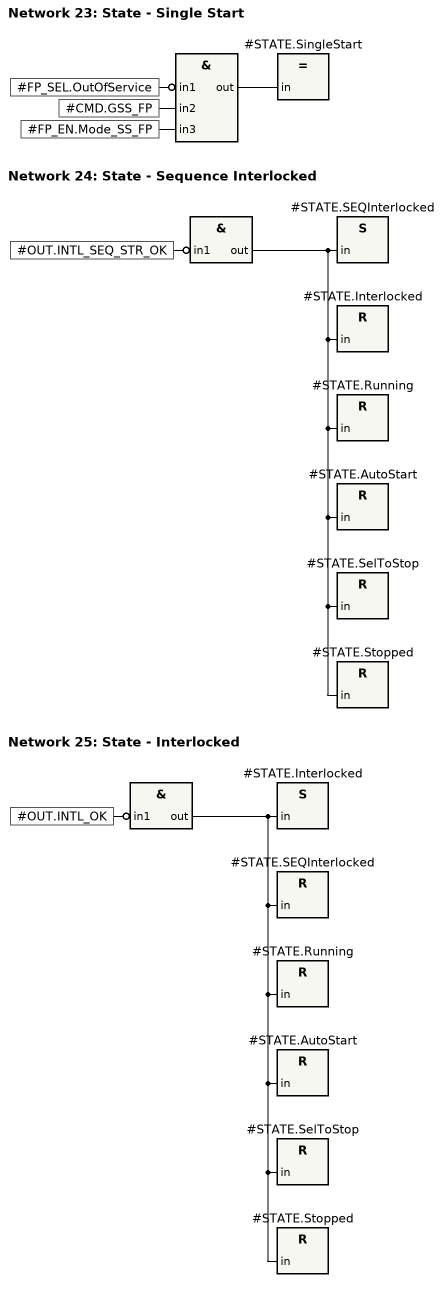
   #STATE.SingleStart := NOT #FP_SEL.OutOfService AND #CMD.GSS_FP AND #FP_EN.Mode_SS_FP;
END_REGION

REGION Network 24: State - Sequence Interlocked
   // Build 3 - SA added
   IF NOT #OUT.INTL_SEQ_STR_OK THEN
       #STATE.SEQInterlocked := TRUE;
       #STATE.Interlocked := FALSE;
       #STATE.Running := FALSE;
       #STATE.AutoStart := FALSE;
       #STATE.SelToStop := FALSE;
       #STATE.Stopped := FALSE;
   END_IF;
END_REGION

REGION Network 25: State - Interlocked
   IF NOT #OUT.INTL_OK THEN
       #STATE.Interlocked := TRUE;
       #STATE.SEQInterlocked := FALSE;
       #STATE.Running := FALSE;
       #STATE.AutoStart := FALSE;
       #STATE.SelToStop := FALSE;
       #STATE.Stopped := FALSE;
   END_IF;
END_REGION

REGION Network 26: Set Output Command for Programs
   // Start command
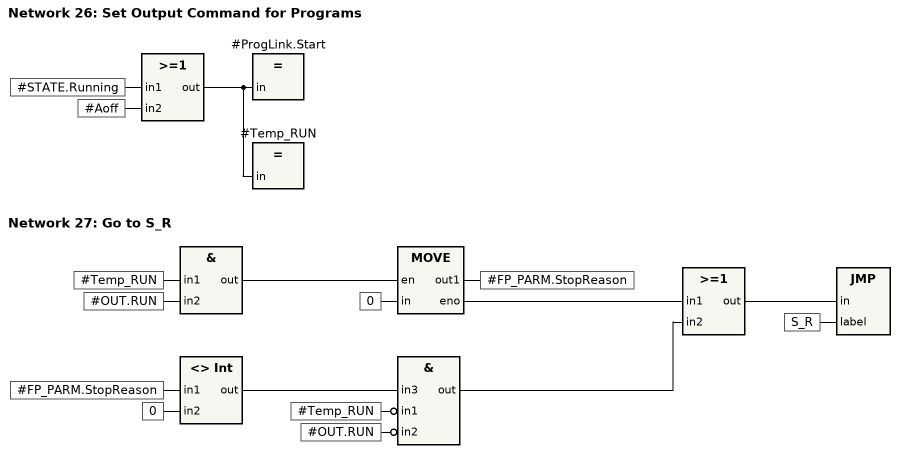
   #ProgLink.Start := #STATE.Running OR #Aoff;
   #Temp_RUN := #ProgLink.Start;
END_REGION

REGION Network 27: Go to S_R
   // ENO of a box is taken as its EN; it also drops when the box reports an error
   #_w1 := #Temp_RUN AND #OUT.RUN;
   IF #_w1 THEN #FP_PARM.StopReason := 0; END_IF;
   IF #_w1 OR ((#FP_PARM.StopReason <> 0) AND NOT #Temp_RUN AND NOT #OUT.RUN) THEN GOTO S_R; END_IF;
END_REGION

REGION Network 28: Stop Reason
   // 0=In Operation
   // 1=Normal Stop
   // 2=Quick Stop
   // 3=Faceplate Stop
   // 6=Quick Stop From Unit Faceplate
   // 9=Sequence Interlock
   // 10=Interlock
   // 12=Emergency Stop
   // 13=Auto Start
   // 99=Unknown Reason
   // 
   // 
   // Build 003-11 Aug 2021- SURAM-IN- Interval Start Stop Reason Added
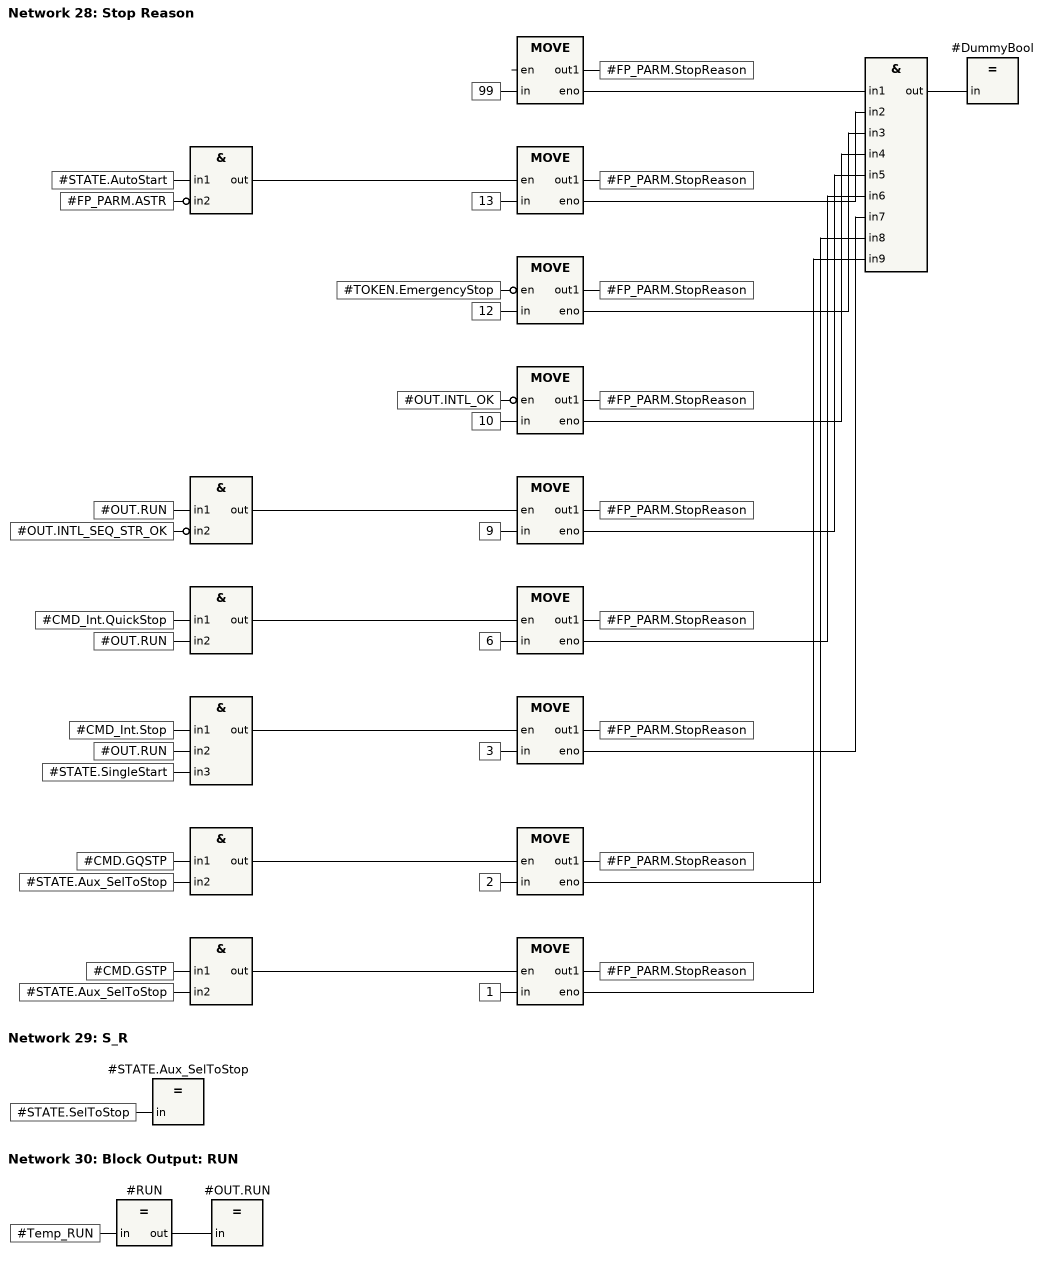
   // ENO of a box is taken as its EN; it also drops when the box reports an error
   #FP_PARM.StopReason := 99;
   #_w1 := #STATE.AutoStart AND NOT #FP_PARM.ASTR;
   IF #_w1 THEN #FP_PARM.StopReason := 13; END_IF;
   IF NOT #TOKEN.EmergencyStop THEN #FP_PARM.StopReason := 12; END_IF;
   IF NOT #OUT.INTL_OK THEN #FP_PARM.StopReason := 10; END_IF;
   #_w2 := #OUT.RUN AND NOT #OUT.INTL_SEQ_STR_OK;
   IF #_w2 THEN #FP_PARM.StopReason := 9; END_IF;
   #_w3 := #CMD_Int.QuickStop AND #OUT.RUN;
   IF #_w3 THEN #FP_PARM.StopReason := 6; END_IF;
   #_w4 := #CMD_Int.Stop AND #OUT.RUN AND #STATE.SingleStart;
   IF #_w4 THEN #FP_PARM.StopReason := 3; END_IF;
   #_w5 := #CMD.GQSTP AND #STATE.Aux_SelToStop;
   IF #_w5 THEN #FP_PARM.StopReason := 2; END_IF;
   #_w6 := #CMD.GSTP AND #STATE.Aux_SelToStop;
   IF #_w6 THEN #FP_PARM.StopReason := 1; END_IF;
   #DummyBool := #_w1 AND NOT #TOKEN.EmergencyStop AND NOT #OUT.INTL_OK AND #_w2 AND #_w3 AND #_w4 AND #_w5 AND #_w6;
END_REGION

REGION Network 29: S_R
   S_R:
   #STATE.Aux_SelToStop := #STATE.SelToStop;
END_REGION

REGION Network 30: Block Output: RUN
   #RUN := #Temp_RUN;
   #OUT.RUN := #Temp_RUN;
END_REGION

REGION Network 31: Reset Commands
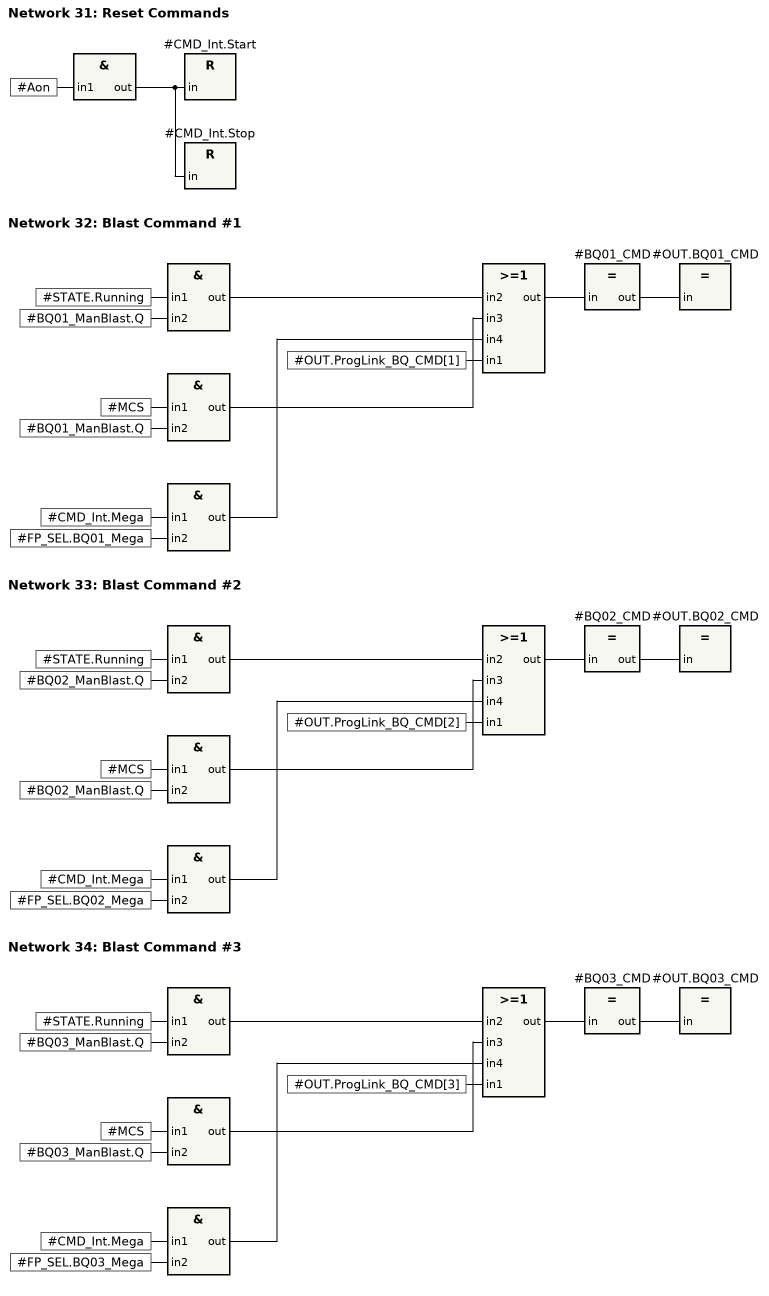
   IF #Aon THEN
       #CMD_Int.Start := FALSE;
       #CMD_Int.Stop := FALSE;
   END_IF;
END_REGION

REGION Network 32: Blast Command #1
   #BQ01_CMD := (#STATE.Running AND #BQ01_ManBlast.Q) OR (#MCS AND #BQ01_ManBlast.Q) OR (#CMD_Int.Mega AND #FP_SEL.BQ01_Mega) OR #OUT.ProgLink_BQ_CMD[1];
   #OUT.BQ01_CMD := #BQ01_CMD;
END_REGION

REGION Network 33: Blast Command #2
   #BQ02_CMD := (#STATE.Running AND #BQ02_ManBlast.Q) OR (#MCS AND #BQ02_ManBlast.Q) OR (#CMD_Int.Mega AND #FP_SEL.BQ02_Mega) OR #OUT.ProgLink_BQ_CMD[2];
   #OUT.BQ02_CMD := #BQ02_CMD;
END_REGION

REGION Network 34: Blast Command #3
   #BQ03_CMD := (#STATE.Running AND #BQ03_ManBlast.Q) OR (#MCS AND #BQ03_ManBlast.Q) OR (#CMD_Int.Mega AND #FP_SEL.BQ03_Mega) OR #OUT.ProgLink_BQ_CMD[3];
   #OUT.BQ03_CMD := #BQ03_CMD;
END_REGION

REGION Network 35: Blast Command #4
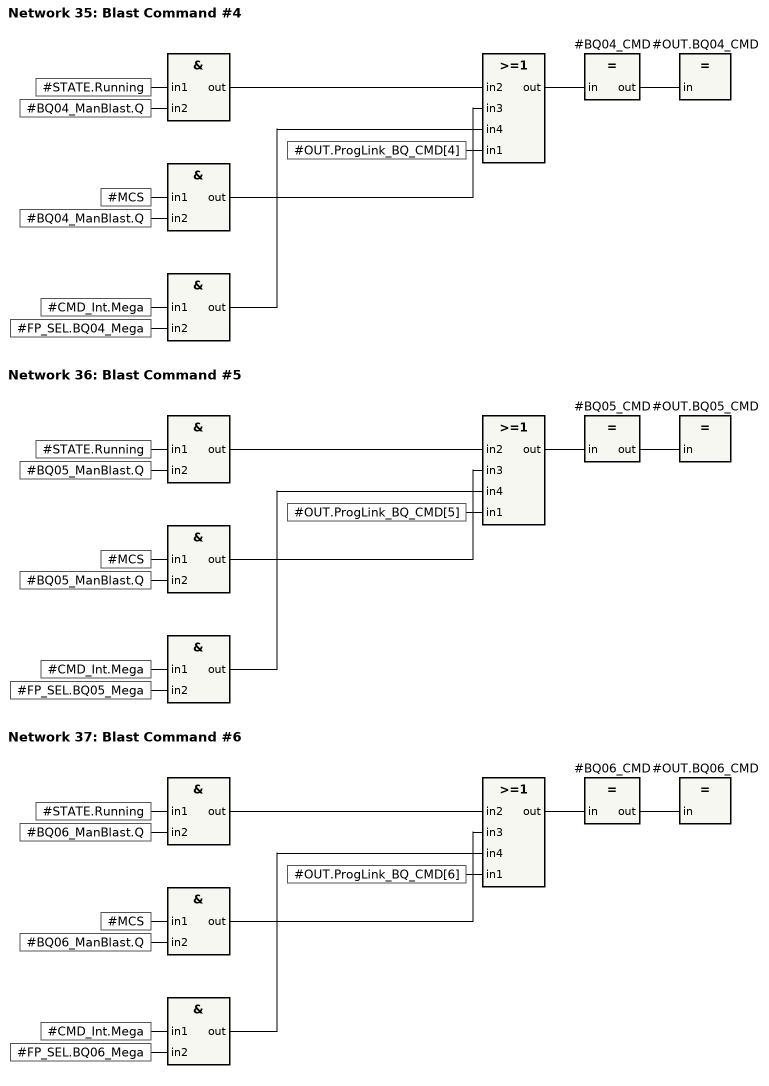
   #BQ04_CMD := (#STATE.Running AND #BQ04_ManBlast.Q) OR (#MCS AND #BQ04_ManBlast.Q) OR (#CMD_Int.Mega AND #FP_SEL.BQ04_Mega) OR #OUT.ProgLink_BQ_CMD[4];
   #OUT.BQ04_CMD := #BQ04_CMD;
END_REGION

REGION Network 36: Blast Command #5
   #BQ05_CMD := (#STATE.Running AND #BQ05_ManBlast.Q) OR (#MCS AND #BQ05_ManBlast.Q) OR (#CMD_Int.Mega AND #FP_SEL.BQ05_Mega) OR #OUT.ProgLink_BQ_CMD[5];
   #OUT.BQ05_CMD := #BQ05_CMD;
END_REGION

REGION Network 37: Blast Command #6
   #BQ06_CMD := (#STATE.Running AND #BQ06_ManBlast.Q) OR (#MCS AND #BQ06_ManBlast.Q) OR (#CMD_Int.Mega AND #FP_SEL.BQ06_Mega) OR #OUT.ProgLink_BQ_CMD[6];
   #OUT.BQ06_CMD := #BQ06_CMD;
END_REGION

REGION Network 38: Blast Command #7
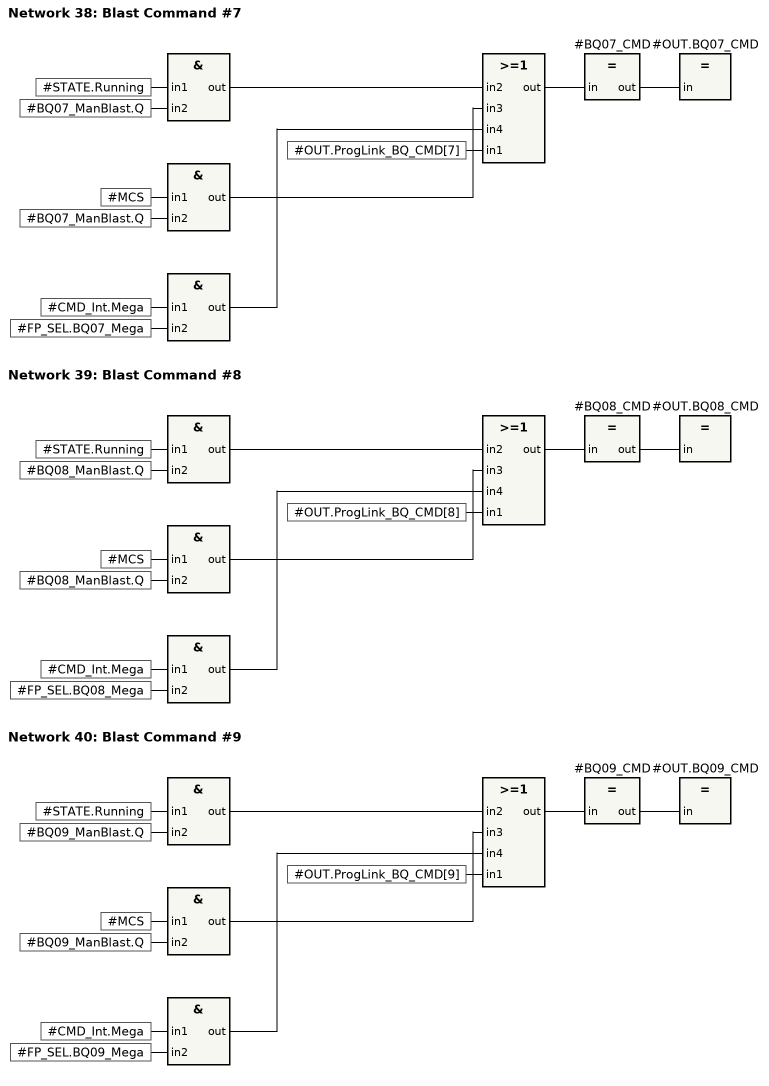
   #BQ07_CMD := (#STATE.Running AND #BQ07_ManBlast.Q) OR (#MCS AND #BQ07_ManBlast.Q) OR (#CMD_Int.Mega AND #FP_SEL.BQ07_Mega) OR #OUT.ProgLink_BQ_CMD[7];
   #OUT.BQ07_CMD := #BQ07_CMD;
END_REGION

REGION Network 39: Blast Command #8
   #BQ08_CMD := (#STATE.Running AND #BQ08_ManBlast.Q) OR (#MCS AND #BQ08_ManBlast.Q) OR (#CMD_Int.Mega AND #FP_SEL.BQ08_Mega) OR #OUT.ProgLink_BQ_CMD[8];
   #OUT.BQ08_CMD := #BQ08_CMD;
END_REGION

REGION Network 40: Blast Command #9
   #BQ09_CMD := (#STATE.Running AND #BQ09_ManBlast.Q) OR (#MCS AND #BQ09_ManBlast.Q) OR (#CMD_Int.Mega AND #FP_SEL.BQ09_Mega) OR #OUT.ProgLink_BQ_CMD[9];
   #OUT.BQ09_CMD := #BQ09_CMD;
END_REGION

REGION Network 41: Blast Command #10
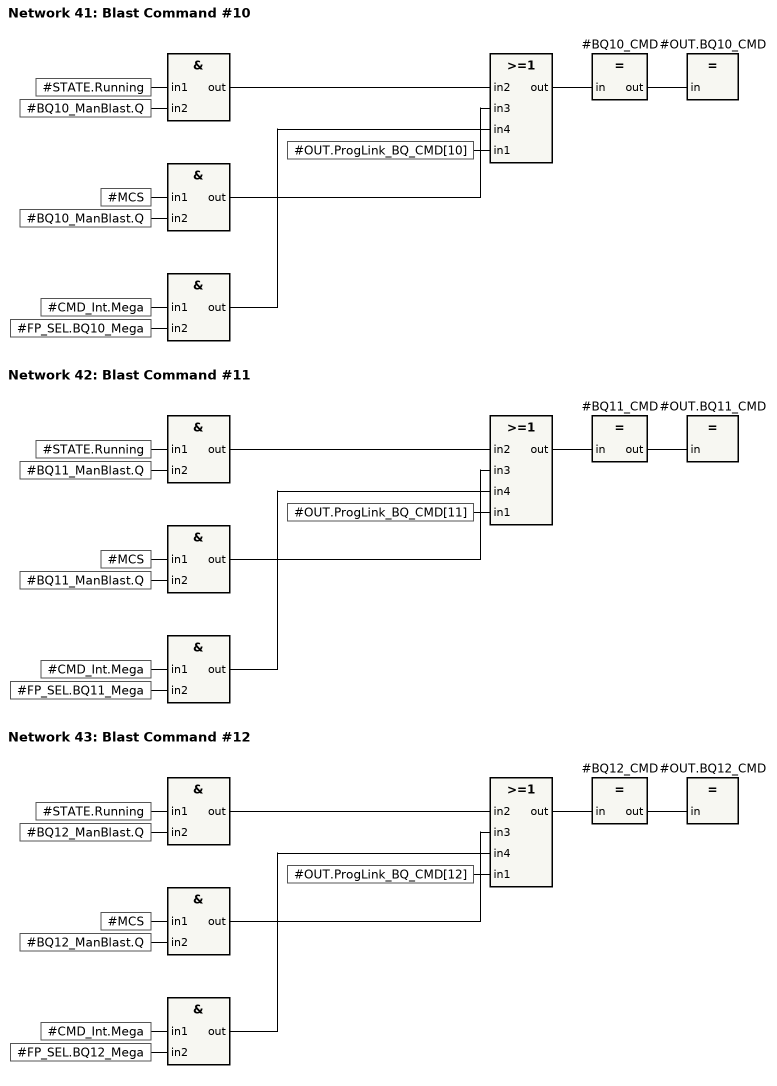
   #BQ10_CMD := (#STATE.Running AND #BQ10_ManBlast.Q) OR (#MCS AND #BQ10_ManBlast.Q) OR (#CMD_Int.Mega AND #FP_SEL.BQ10_Mega) OR #OUT.ProgLink_BQ_CMD[10];
   #OUT.BQ10_CMD := #BQ10_CMD;
END_REGION

REGION Network 42: Blast Command #11
   #BQ11_CMD := (#STATE.Running AND #BQ11_ManBlast.Q) OR (#MCS AND #BQ11_ManBlast.Q) OR (#CMD_Int.Mega AND #FP_SEL.BQ11_Mega) OR #OUT.ProgLink_BQ_CMD[11];
   #OUT.BQ11_CMD := #BQ11_CMD;
END_REGION

REGION Network 43: Blast Command #12
   #BQ12_CMD := (#STATE.Running AND #BQ12_ManBlast.Q) OR (#MCS AND #BQ12_ManBlast.Q) OR (#CMD_Int.Mega AND #FP_SEL.BQ12_Mega) OR #OUT.ProgLink_BQ_CMD[12];
   #OUT.BQ12_CMD := #BQ12_CMD;
END_REGION

REGION Network 44: Blast Command #13
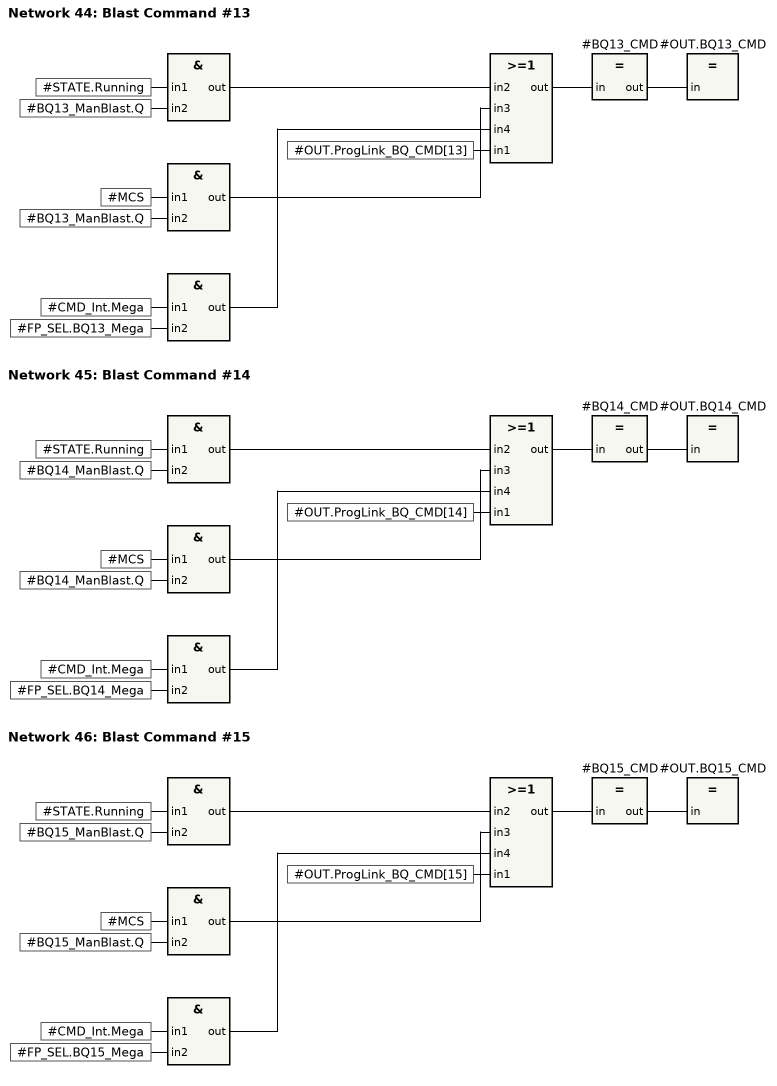
   #BQ13_CMD := (#STATE.Running AND #BQ13_ManBlast.Q) OR (#MCS AND #BQ13_ManBlast.Q) OR (#CMD_Int.Mega AND #FP_SEL.BQ13_Mega) OR #OUT.ProgLink_BQ_CMD[13];
   #OUT.BQ13_CMD := #BQ13_CMD;
END_REGION

REGION Network 45: Blast Command #14
   #BQ14_CMD := (#STATE.Running AND #BQ14_ManBlast.Q) OR (#MCS AND #BQ14_ManBlast.Q) OR (#CMD_Int.Mega AND #FP_SEL.BQ14_Mega) OR #OUT.ProgLink_BQ_CMD[14];
   #OUT.BQ14_CMD := #BQ14_CMD;
END_REGION

REGION Network 46: Blast Command #15
   #BQ15_CMD := (#STATE.Running AND #BQ15_ManBlast.Q) OR (#MCS AND #BQ15_ManBlast.Q) OR (#CMD_Int.Mega AND #FP_SEL.BQ15_Mega) OR #OUT.ProgLink_BQ_CMD[15];
   #OUT.BQ15_CMD := #BQ15_CMD;
END_REGION

REGION Network 47: Blast Command #16
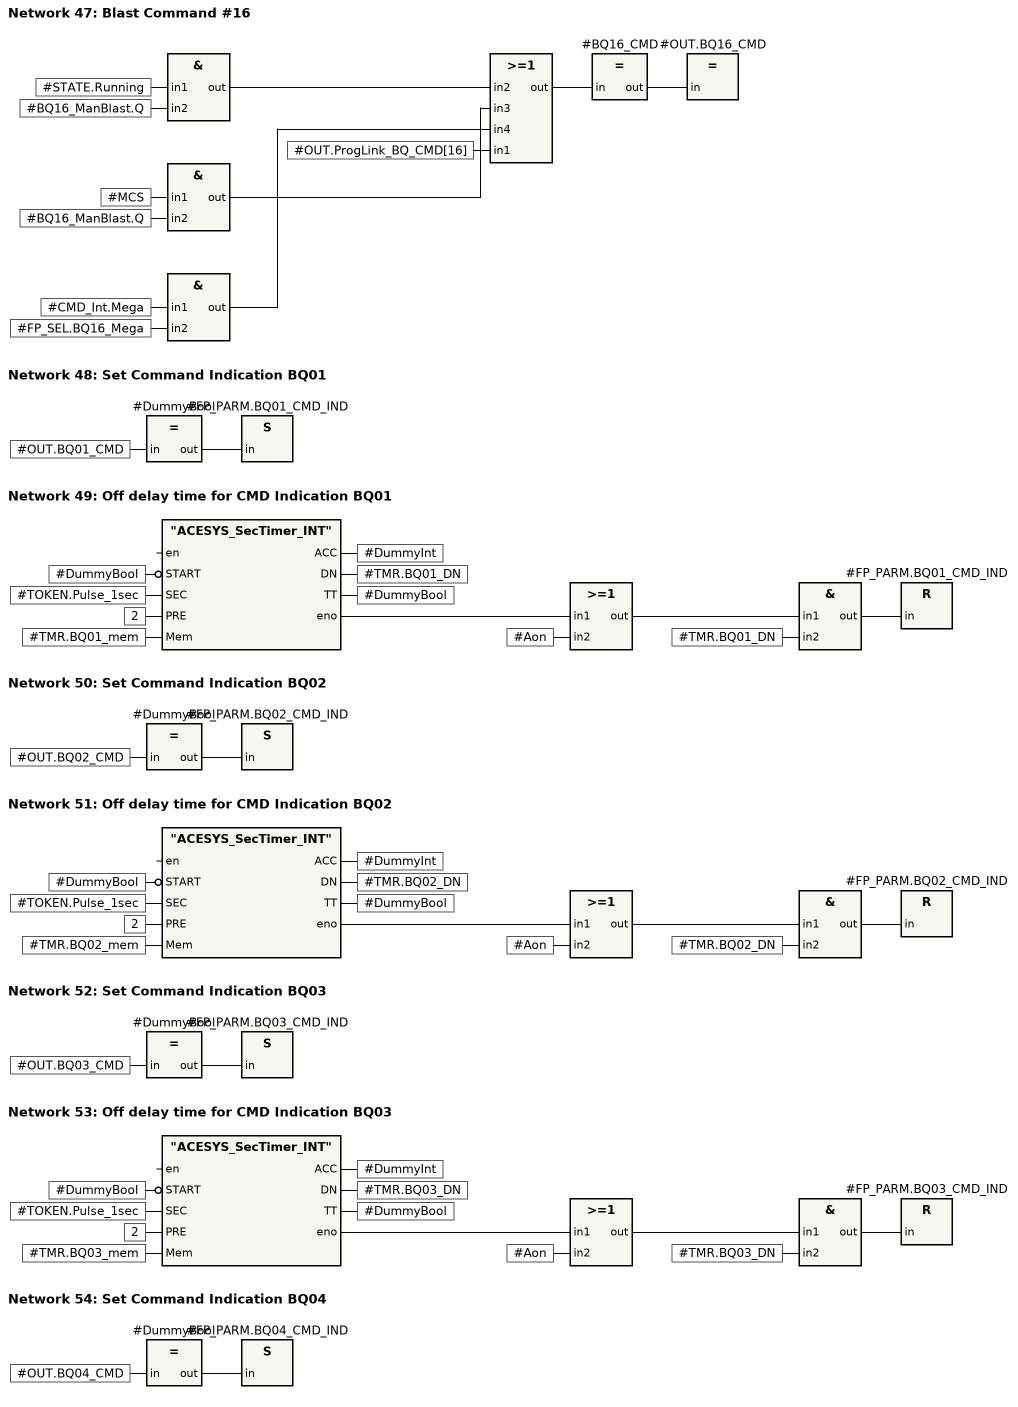
   #BQ16_CMD := (#STATE.Running AND #BQ16_ManBlast.Q) OR (#MCS AND #BQ16_ManBlast.Q) OR (#CMD_Int.Mega AND #FP_SEL.BQ16_Mega) OR #OUT.ProgLink_BQ_CMD[16];
   #OUT.BQ16_CMD := #BQ16_CMD;
END_REGION

REGION Network 48: Set Command Indication BQ01
   // Build 2 New NW
   #DummyBool := #OUT.BQ01_CMD;
   IF #OUT.BQ01_CMD THEN #FP_PARM.BQ01_CMD_IND := TRUE; END_IF;
END_REGION

REGION Network 49: Off delay time for CMD Indication BQ01
   // Build 2 New NW
   "ACESYS_SecTimer_INT"(START := NOT #DummyBool,
                         SEC := #TOKEN.Pulse_1sec,
                         PRE := 2,
                         Mem := #TMR.BQ01_mem,
                         ACC => #DummyInt,
                         DN => #TMR.BQ01_DN,
                         TT => #DummyBool,
                         ENO => #_w1);
   IF (#_w1 OR #Aon) AND #TMR.BQ01_DN THEN #FP_PARM.BQ01_CMD_IND := FALSE; END_IF;
END_REGION

REGION Network 50: Set Command Indication BQ02
   // Build 2 New NW
   #DummyBool := #OUT.BQ02_CMD;
   IF #OUT.BQ02_CMD THEN #FP_PARM.BQ02_CMD_IND := TRUE; END_IF;
END_REGION

REGION Network 51: Off delay time for CMD Indication BQ02
   // Build 2 New NW
   "ACESYS_SecTimer_INT"(START := NOT #DummyBool,
                         SEC := #TOKEN.Pulse_1sec,
                         PRE := 2,
                         Mem := #TMR.BQ02_mem,
                         ACC => #DummyInt,
                         DN => #TMR.BQ02_DN,
                         TT => #DummyBool,
                         ENO => #_w1);
   IF (#_w1 OR #Aon) AND #TMR.BQ02_DN THEN #FP_PARM.BQ02_CMD_IND := FALSE; END_IF;
END_REGION

REGION Network 52: Set Command Indication BQ03
   // Build 2 New NW
   #DummyBool := #OUT.BQ03_CMD;
   IF #OUT.BQ03_CMD THEN #FP_PARM.BQ03_CMD_IND := TRUE; END_IF;
END_REGION

REGION Network 53: Off delay time for CMD Indication BQ03
   // Build 2 New NW
   "ACESYS_SecTimer_INT"(START := NOT #DummyBool,
                         SEC := #TOKEN.Pulse_1sec,
                         PRE := 2,
                         Mem := #TMR.BQ03_mem,
                         ACC => #DummyInt,
                         DN => #TMR.BQ03_DN,
                         TT => #DummyBool,
                         ENO => #_w1);
   IF (#_w1 OR #Aon) AND #TMR.BQ03_DN THEN #FP_PARM.BQ03_CMD_IND := FALSE; END_IF;
END_REGION

REGION Network 54: Set Command Indication BQ04
   // Build 2 New NW
   #DummyBool := #OUT.BQ04_CMD;
   IF #OUT.BQ04_CMD THEN #FP_PARM.BQ04_CMD_IND := TRUE; END_IF;
END_REGION

REGION Network 55: Off delay time for CMD Indication BQ04
   // Build 2 New NW
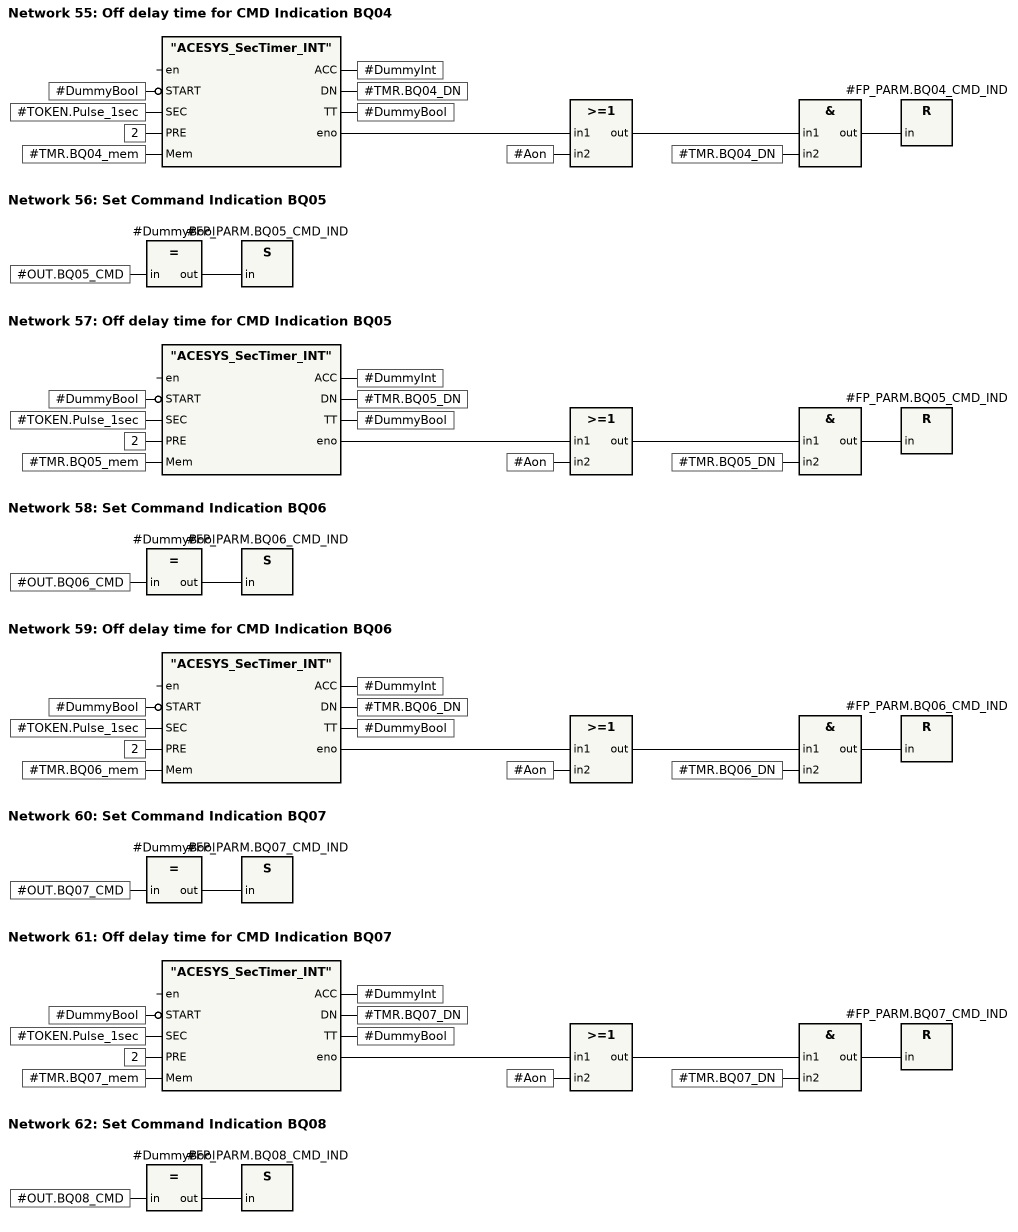
   "ACESYS_SecTimer_INT"(START := NOT #DummyBool,
                         SEC := #TOKEN.Pulse_1sec,
                         PRE := 2,
                         Mem := #TMR.BQ04_mem,
                         ACC => #DummyInt,
                         DN => #TMR.BQ04_DN,
                         TT => #DummyBool,
                         ENO => #_w1);
   IF (#_w1 OR #Aon) AND #TMR.BQ04_DN THEN #FP_PARM.BQ04_CMD_IND := FALSE; END_IF;
END_REGION

REGION Network 56: Set Command Indication BQ05
   // Build 2 New NW
   #DummyBool := #OUT.BQ05_CMD;
   IF #OUT.BQ05_CMD THEN #FP_PARM.BQ05_CMD_IND := TRUE; END_IF;
END_REGION

REGION Network 57: Off delay time for CMD Indication BQ05
   // Build 2 New NW
   "ACESYS_SecTimer_INT"(START := NOT #DummyBool,
                         SEC := #TOKEN.Pulse_1sec,
                         PRE := 2,
                         Mem := #TMR.BQ05_mem,
                         ACC => #DummyInt,
                         DN => #TMR.BQ05_DN,
                         TT => #DummyBool,
                         ENO => #_w1);
   IF (#_w1 OR #Aon) AND #TMR.BQ05_DN THEN #FP_PARM.BQ05_CMD_IND := FALSE; END_IF;
END_REGION

REGION Network 58: Set Command Indication BQ06
   // Build 2 New NW
   #DummyBool := #OUT.BQ06_CMD;
   IF #OUT.BQ06_CMD THEN #FP_PARM.BQ06_CMD_IND := TRUE; END_IF;
END_REGION

REGION Network 59: Off delay time for CMD Indication BQ06
   // Build 2 New NW
   "ACESYS_SecTimer_INT"(START := NOT #DummyBool,
                         SEC := #TOKEN.Pulse_1sec,
                         PRE := 2,
                         Mem := #TMR.BQ06_mem,
                         ACC => #DummyInt,
                         DN => #TMR.BQ06_DN,
                         TT => #DummyBool,
                         ENO => #_w1);
   IF (#_w1 OR #Aon) AND #TMR.BQ06_DN THEN #FP_PARM.BQ06_CMD_IND := FALSE; END_IF;
END_REGION

REGION Network 60: Set Command Indication BQ07
   // Build 2 New NW
   #DummyBool := #OUT.BQ07_CMD;
   IF #OUT.BQ07_CMD THEN #FP_PARM.BQ07_CMD_IND := TRUE; END_IF;
END_REGION

REGION Network 61: Off delay time for CMD Indication BQ07
   // Build 2 New NW
   "ACESYS_SecTimer_INT"(START := NOT #DummyBool,
                         SEC := #TOKEN.Pulse_1sec,
                         PRE := 2,
                         Mem := #TMR.BQ07_mem,
                         ACC => #DummyInt,
                         DN => #TMR.BQ07_DN,
                         TT => #DummyBool,
                         ENO => #_w1);
   IF (#_w1 OR #Aon) AND #TMR.BQ07_DN THEN #FP_PARM.BQ07_CMD_IND := FALSE; END_IF;
END_REGION

REGION Network 62: Set Command Indication BQ08
   // Build 2 New NW
   #DummyBool := #OUT.BQ08_CMD;
   IF #OUT.BQ08_CMD THEN #FP_PARM.BQ08_CMD_IND := TRUE; END_IF;
END_REGION

REGION Network 63: Off delay time for CMD Indication BQ08
   // Build 2 New NW
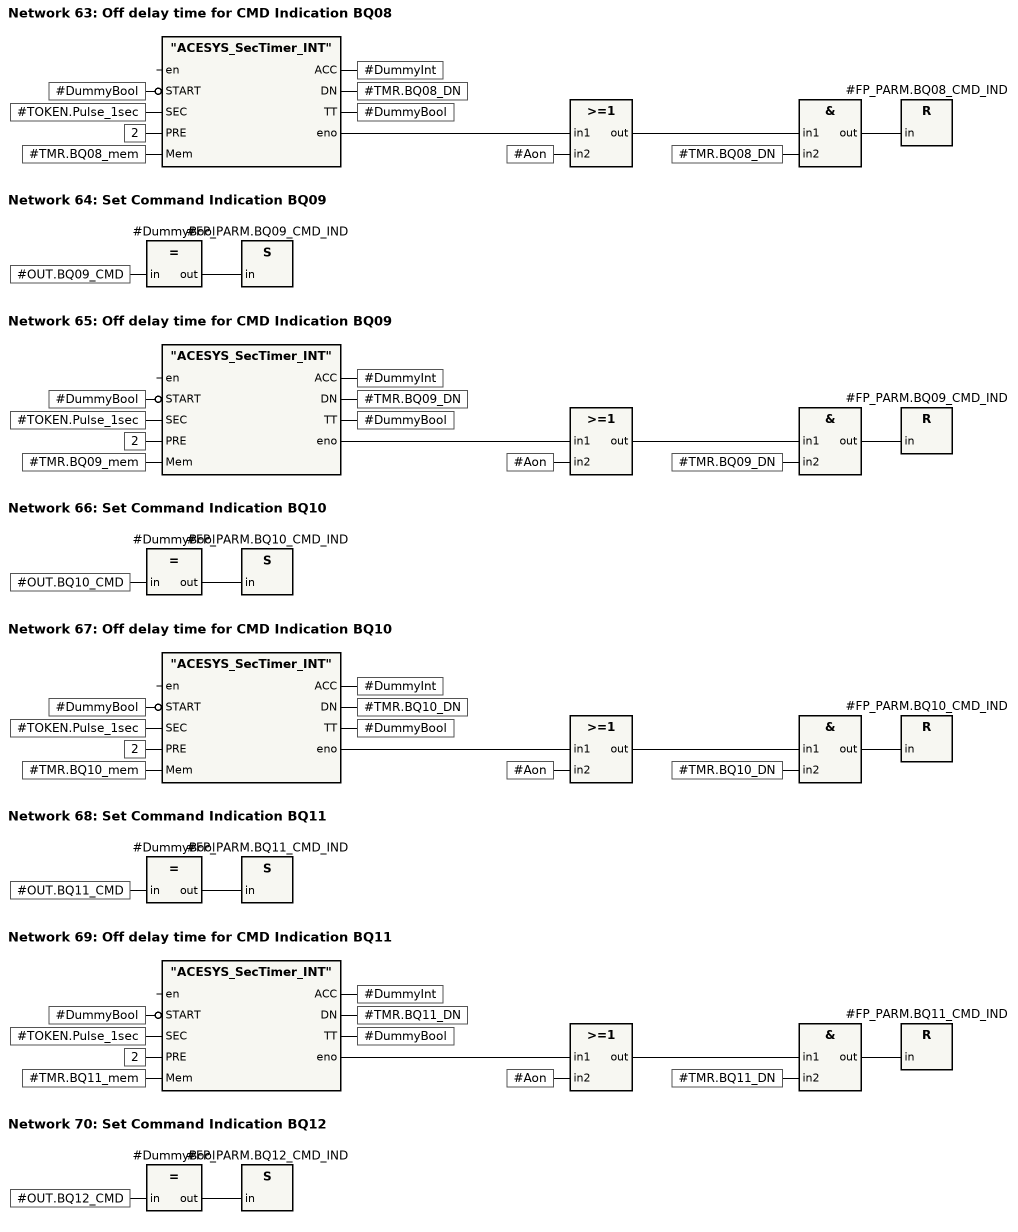
   "ACESYS_SecTimer_INT"(START := NOT #DummyBool,
                         SEC := #TOKEN.Pulse_1sec,
                         PRE := 2,
                         Mem := #TMR.BQ08_mem,
                         ACC => #DummyInt,
                         DN => #TMR.BQ08_DN,
                         TT => #DummyBool,
                         ENO => #_w1);
   IF (#_w1 OR #Aon) AND #TMR.BQ08_DN THEN #FP_PARM.BQ08_CMD_IND := FALSE; END_IF;
END_REGION

REGION Network 64: Set Command Indication BQ09
   // Build 2 New NW
   #DummyBool := #OUT.BQ09_CMD;
   IF #OUT.BQ09_CMD THEN #FP_PARM.BQ09_CMD_IND := TRUE; END_IF;
END_REGION

REGION Network 65: Off delay time for CMD Indication BQ09
   // Build 2 New NW
   "ACESYS_SecTimer_INT"(START := NOT #DummyBool,
                         SEC := #TOKEN.Pulse_1sec,
                         PRE := 2,
                         Mem := #TMR.BQ09_mem,
                         ACC => #DummyInt,
                         DN => #TMR.BQ09_DN,
                         TT => #DummyBool,
                         ENO => #_w1);
   IF (#_w1 OR #Aon) AND #TMR.BQ09_DN THEN #FP_PARM.BQ09_CMD_IND := FALSE; END_IF;
END_REGION

REGION Network 66: Set Command Indication BQ10
   // Build 2 New NW
   #DummyBool := #OUT.BQ10_CMD;
   IF #OUT.BQ10_CMD THEN #FP_PARM.BQ10_CMD_IND := TRUE; END_IF;
END_REGION

REGION Network 67: Off delay time for CMD Indication BQ10
   // Build 2 New NW
   "ACESYS_SecTimer_INT"(START := NOT #DummyBool,
                         SEC := #TOKEN.Pulse_1sec,
                         PRE := 2,
                         Mem := #TMR.BQ10_mem,
                         ACC => #DummyInt,
                         DN => #TMR.BQ10_DN,
                         TT => #DummyBool,
                         ENO => #_w1);
   IF (#_w1 OR #Aon) AND #TMR.BQ10_DN THEN #FP_PARM.BQ10_CMD_IND := FALSE; END_IF;
END_REGION

REGION Network 68: Set Command Indication BQ11
   // Build 2 New NW
   #DummyBool := #OUT.BQ11_CMD;
   IF #OUT.BQ11_CMD THEN #FP_PARM.BQ11_CMD_IND := TRUE; END_IF;
END_REGION

REGION Network 69: Off delay time for CMD Indication BQ11
   // Build 2 New NW
   "ACESYS_SecTimer_INT"(START := NOT #DummyBool,
                         SEC := #TOKEN.Pulse_1sec,
                         PRE := 2,
                         Mem := #TMR.BQ11_mem,
                         ACC => #DummyInt,
                         DN => #TMR.BQ11_DN,
                         TT => #DummyBool,
                         ENO => #_w1);
   IF (#_w1 OR #Aon) AND #TMR.BQ11_DN THEN #FP_PARM.BQ11_CMD_IND := FALSE; END_IF;
END_REGION

REGION Network 70: Set Command Indication BQ12
   // Build 2 New NW
   #DummyBool := #OUT.BQ12_CMD;
   IF #OUT.BQ12_CMD THEN #FP_PARM.BQ12_CMD_IND := TRUE; END_IF;
END_REGION

REGION Network 71: Off delay time for CMD Indication BQ12
   // Build 2 New NW
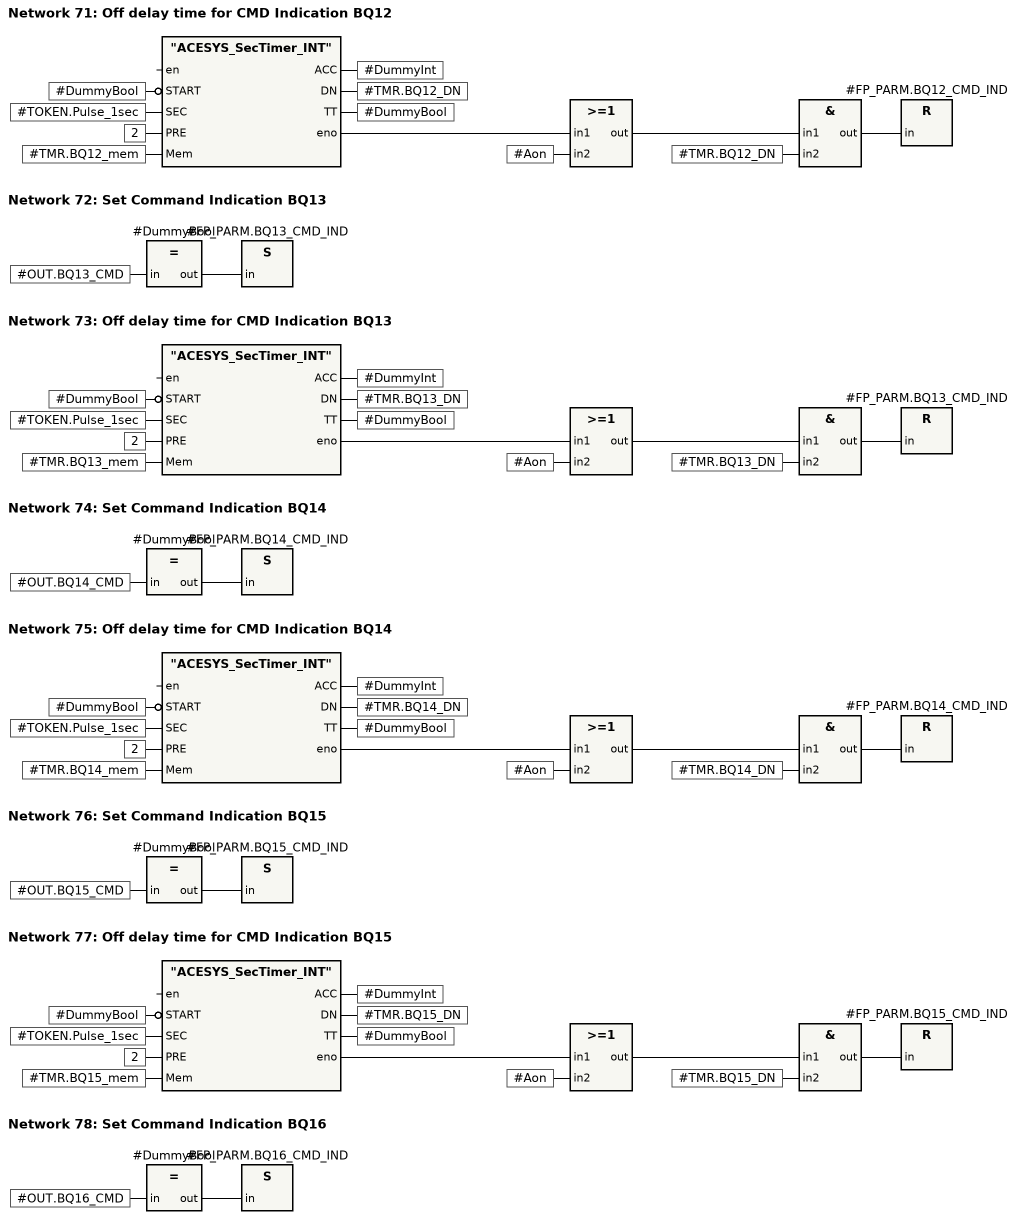
   "ACESYS_SecTimer_INT"(START := NOT #DummyBool,
                         SEC := #TOKEN.Pulse_1sec,
                         PRE := 2,
                         Mem := #TMR.BQ12_mem,
                         ACC => #DummyInt,
                         DN => #TMR.BQ12_DN,
                         TT => #DummyBool,
                         ENO => #_w1);
   IF (#_w1 OR #Aon) AND #TMR.BQ12_DN THEN #FP_PARM.BQ12_CMD_IND := FALSE; END_IF;
END_REGION

REGION Network 72: Set Command Indication BQ13
   // Build 2 New NW
   #DummyBool := #OUT.BQ13_CMD;
   IF #OUT.BQ13_CMD THEN #FP_PARM.BQ13_CMD_IND := TRUE; END_IF;
END_REGION

REGION Network 73: Off delay time for CMD Indication BQ13
   // Build 2 New NW
   "ACESYS_SecTimer_INT"(START := NOT #DummyBool,
                         SEC := #TOKEN.Pulse_1sec,
                         PRE := 2,
                         Mem := #TMR.BQ13_mem,
                         ACC => #DummyInt,
                         DN => #TMR.BQ13_DN,
                         TT => #DummyBool,
                         ENO => #_w1);
   IF (#_w1 OR #Aon) AND #TMR.BQ13_DN THEN #FP_PARM.BQ13_CMD_IND := FALSE; END_IF;
END_REGION

REGION Network 74: Set Command Indication BQ14
   // Build 2 New NW
   #DummyBool := #OUT.BQ14_CMD;
   IF #OUT.BQ14_CMD THEN #FP_PARM.BQ14_CMD_IND := TRUE; END_IF;
END_REGION

REGION Network 75: Off delay time for CMD Indication BQ14
   // Build 2 New NW
   "ACESYS_SecTimer_INT"(START := NOT #DummyBool,
                         SEC := #TOKEN.Pulse_1sec,
                         PRE := 2,
                         Mem := #TMR.BQ14_mem,
                         ACC => #DummyInt,
                         DN => #TMR.BQ14_DN,
                         TT => #DummyBool,
                         ENO => #_w1);
   IF (#_w1 OR #Aon) AND #TMR.BQ14_DN THEN #FP_PARM.BQ14_CMD_IND := FALSE; END_IF;
END_REGION

REGION Network 76: Set Command Indication BQ15
   // Build 2 New NW
   #DummyBool := #OUT.BQ15_CMD;
   IF #OUT.BQ15_CMD THEN #FP_PARM.BQ15_CMD_IND := TRUE; END_IF;
END_REGION

REGION Network 77: Off delay time for CMD Indication BQ15
   // Build 2 New NW
   "ACESYS_SecTimer_INT"(START := NOT #DummyBool,
                         SEC := #TOKEN.Pulse_1sec,
                         PRE := 2,
                         Mem := #TMR.BQ15_mem,
                         ACC => #DummyInt,
                         DN => #TMR.BQ15_DN,
                         TT => #DummyBool,
                         ENO => #_w1);
   IF (#_w1 OR #Aon) AND #TMR.BQ15_DN THEN #FP_PARM.BQ15_CMD_IND := FALSE; END_IF;
END_REGION

REGION Network 78: Set Command Indication BQ16
   // Build 2 New NW
   #DummyBool := #OUT.BQ16_CMD;
   IF #OUT.BQ16_CMD THEN #FP_PARM.BQ16_CMD_IND := TRUE; END_IF;
END_REGION

REGION Network 79: Off delay time for CMD Indication BQ16
   // Build 2 New NW
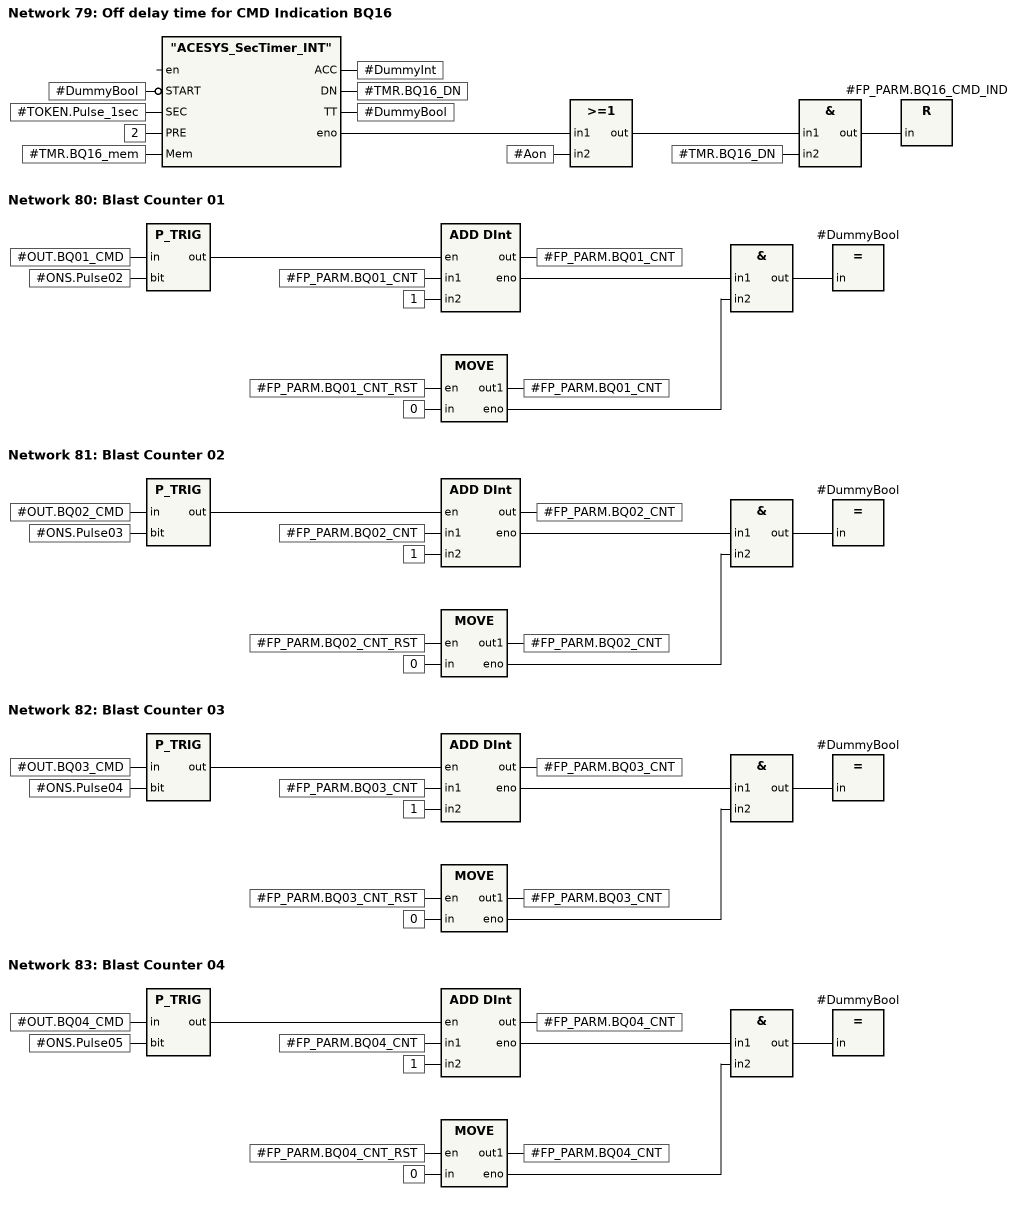
   "ACESYS_SecTimer_INT"(START := NOT #DummyBool,
                         SEC := #TOKEN.Pulse_1sec,
                         PRE := 2,
                         Mem := #TMR.BQ16_mem,
                         ACC => #DummyInt,
                         DN => #TMR.BQ16_DN,
                         TT => #DummyBool,
                         ENO => #_w1);
   IF (#_w1 OR #Aon) AND #TMR.BQ16_DN THEN #FP_PARM.BQ16_CMD_IND := FALSE; END_IF;
END_REGION

REGION Network 80: Blast Counter 01
   // ENO of a box is taken as its EN; it also drops when the box reports an error
   #_w1 := #OUT.BQ01_CMD AND NOT #ONS.Pulse02;   // rising edge
   #ONS.Pulse02 := #OUT.BQ01_CMD;
   IF #_w1 THEN #FP_PARM.BQ01_CNT := #FP_PARM.BQ01_CNT + 1; END_IF;
   IF #FP_PARM.BQ01_CNT_RST THEN #FP_PARM.BQ01_CNT := 0; END_IF;
   #DummyBool := #_w1 AND #FP_PARM.BQ01_CNT_RST;
END_REGION

REGION Network 81: Blast Counter 02
   // ENO of a box is taken as its EN; it also drops when the box reports an error
   #_w1 := #OUT.BQ02_CMD AND NOT #ONS.Pulse03;   // rising edge
   #ONS.Pulse03 := #OUT.BQ02_CMD;
   IF #_w1 THEN #FP_PARM.BQ02_CNT := #FP_PARM.BQ02_CNT + 1; END_IF;
   IF #FP_PARM.BQ02_CNT_RST THEN #FP_PARM.BQ02_CNT := 0; END_IF;
   #DummyBool := #_w1 AND #FP_PARM.BQ02_CNT_RST;
END_REGION

REGION Network 82: Blast Counter 03
   // ENO of a box is taken as its EN; it also drops when the box reports an error
   #_w1 := #OUT.BQ03_CMD AND NOT #ONS.Pulse04;   // rising edge
   #ONS.Pulse04 := #OUT.BQ03_CMD;
   IF #_w1 THEN #FP_PARM.BQ03_CNT := #FP_PARM.BQ03_CNT + 1; END_IF;
   IF #FP_PARM.BQ03_CNT_RST THEN #FP_PARM.BQ03_CNT := 0; END_IF;
   #DummyBool := #_w1 AND #FP_PARM.BQ03_CNT_RST;
END_REGION

REGION Network 83: Blast Counter 04
   // ENO of a box is taken as its EN; it also drops when the box reports an error
   #_w1 := #OUT.BQ04_CMD AND NOT #ONS.Pulse05;   // rising edge
   #ONS.Pulse05 := #OUT.BQ04_CMD;
   IF #_w1 THEN #FP_PARM.BQ04_CNT := #FP_PARM.BQ04_CNT + 1; END_IF;
   IF #FP_PARM.BQ04_CNT_RST THEN #FP_PARM.BQ04_CNT := 0; END_IF;
   #DummyBool := #_w1 AND #FP_PARM.BQ04_CNT_RST;
END_REGION

REGION Network 84: Blast Counter 05
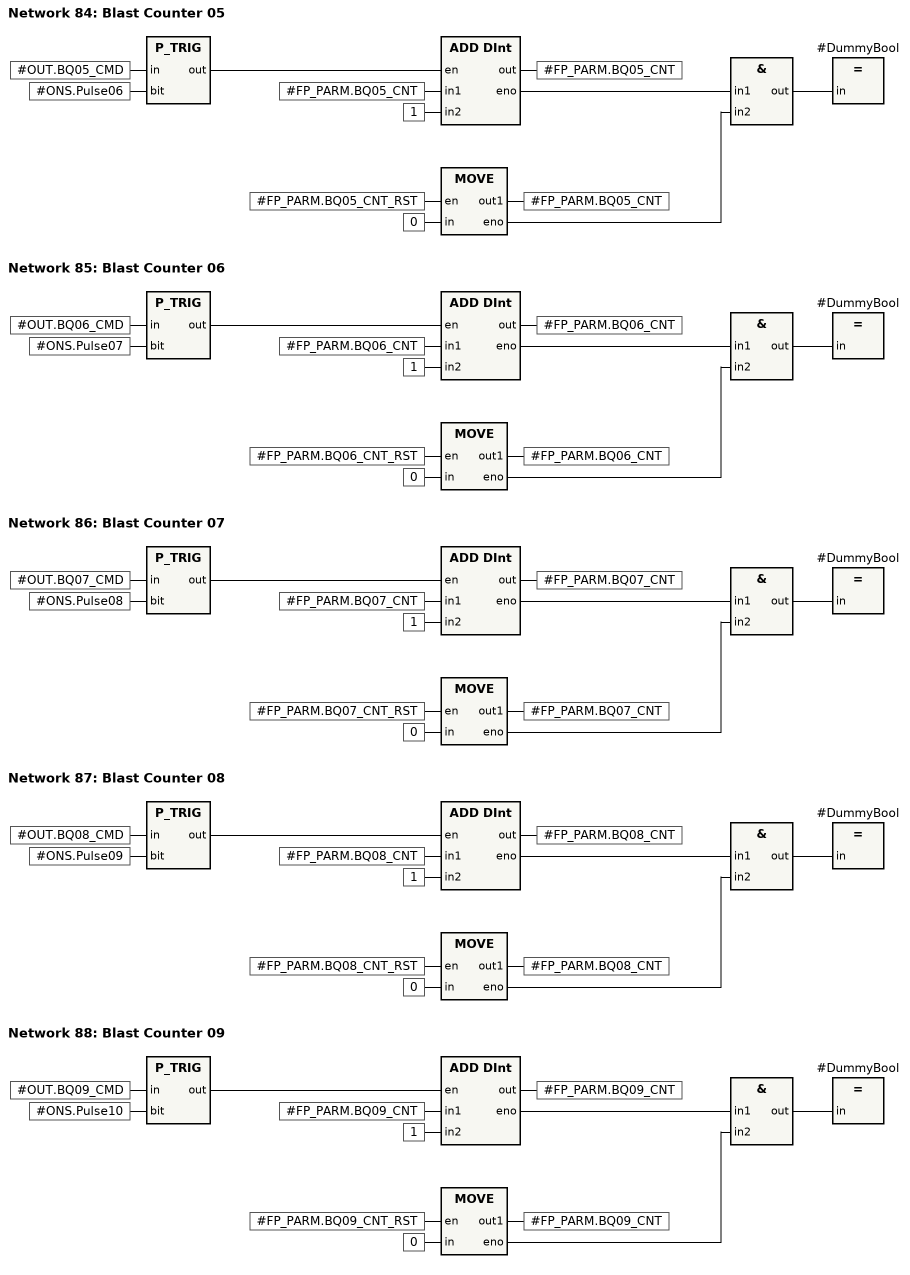
   // ENO of a box is taken as its EN; it also drops when the box reports an error
   #_w1 := #OUT.BQ05_CMD AND NOT #ONS.Pulse06;   // rising edge
   #ONS.Pulse06 := #OUT.BQ05_CMD;
   IF #_w1 THEN #FP_PARM.BQ05_CNT := #FP_PARM.BQ05_CNT + 1; END_IF;
   IF #FP_PARM.BQ05_CNT_RST THEN #FP_PARM.BQ05_CNT := 0; END_IF;
   #DummyBool := #_w1 AND #FP_PARM.BQ05_CNT_RST;
END_REGION

REGION Network 85: Blast Counter 06
   // ENO of a box is taken as its EN; it also drops when the box reports an error
   #_w1 := #OUT.BQ06_CMD AND NOT #ONS.Pulse07;   // rising edge
   #ONS.Pulse07 := #OUT.BQ06_CMD;
   IF #_w1 THEN #FP_PARM.BQ06_CNT := #FP_PARM.BQ06_CNT + 1; END_IF;
   IF #FP_PARM.BQ06_CNT_RST THEN #FP_PARM.BQ06_CNT := 0; END_IF;
   #DummyBool := #_w1 AND #FP_PARM.BQ06_CNT_RST;
END_REGION

REGION Network 86: Blast Counter 07
   // ENO of a box is taken as its EN; it also drops when the box reports an error
   #_w1 := #OUT.BQ07_CMD AND NOT #ONS.Pulse08;   // rising edge
   #ONS.Pulse08 := #OUT.BQ07_CMD;
   IF #_w1 THEN #FP_PARM.BQ07_CNT := #FP_PARM.BQ07_CNT + 1; END_IF;
   IF #FP_PARM.BQ07_CNT_RST THEN #FP_PARM.BQ07_CNT := 0; END_IF;
   #DummyBool := #_w1 AND #FP_PARM.BQ07_CNT_RST;
END_REGION

REGION Network 87: Blast Counter 08
   // ENO of a box is taken as its EN; it also drops when the box reports an error
   #_w1 := #OUT.BQ08_CMD AND NOT #ONS.Pulse09;   // rising edge
   #ONS.Pulse09 := #OUT.BQ08_CMD;
   IF #_w1 THEN #FP_PARM.BQ08_CNT := #FP_PARM.BQ08_CNT + 1; END_IF;
   IF #FP_PARM.BQ08_CNT_RST THEN #FP_PARM.BQ08_CNT := 0; END_IF;
   #DummyBool := #_w1 AND #FP_PARM.BQ08_CNT_RST;
END_REGION

REGION Network 88: Blast Counter 09
   // ENO of a box is taken as its EN; it also drops when the box reports an error
   #_w1 := #OUT.BQ09_CMD AND NOT #ONS.Pulse10;   // rising edge
   #ONS.Pulse10 := #OUT.BQ09_CMD;
   IF #_w1 THEN #FP_PARM.BQ09_CNT := #FP_PARM.BQ09_CNT + 1; END_IF;
   IF #FP_PARM.BQ09_CNT_RST THEN #FP_PARM.BQ09_CNT := 0; END_IF;
   #DummyBool := #_w1 AND #FP_PARM.BQ09_CNT_RST;
END_REGION

REGION Network 89: Blast Counter 10
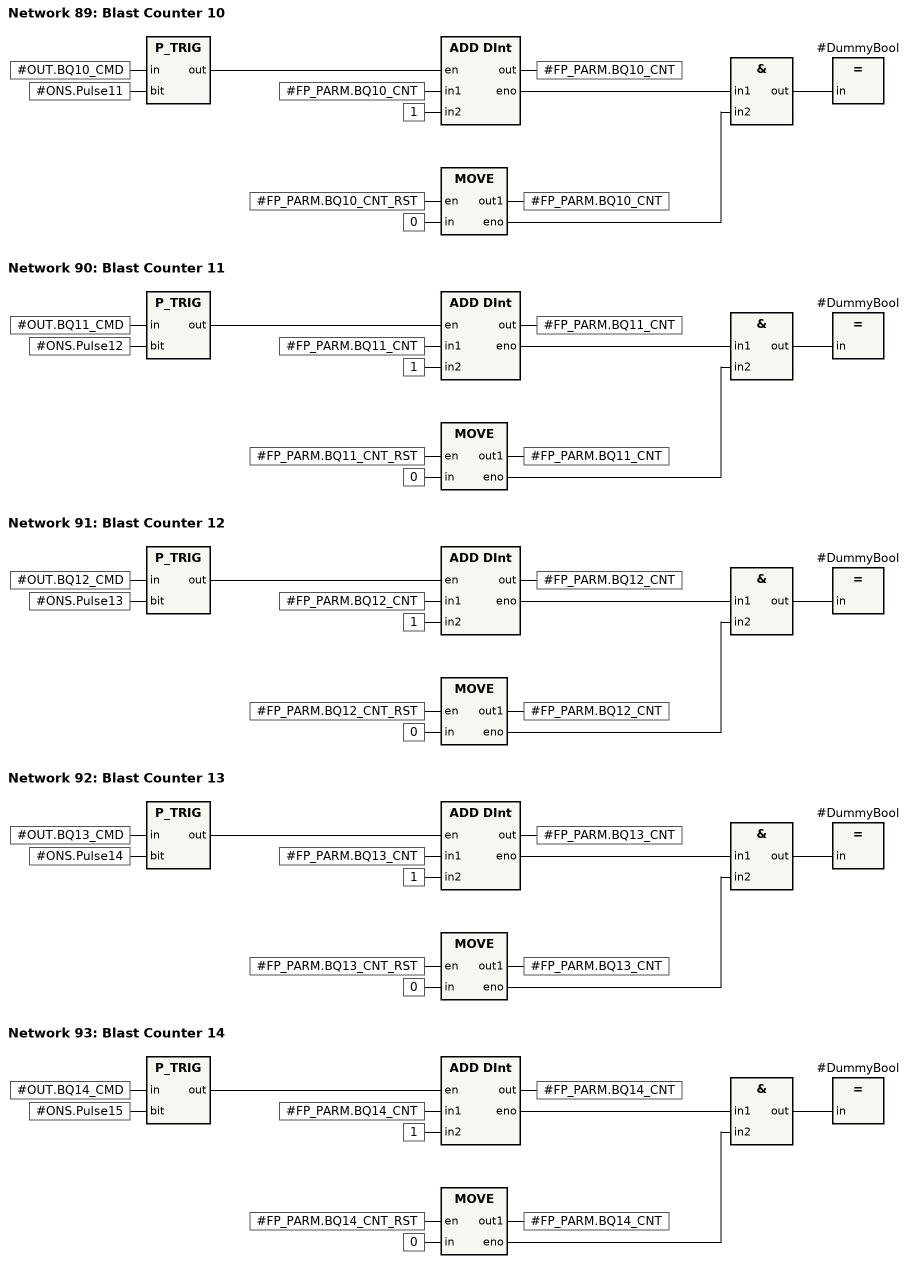
   // ENO of a box is taken as its EN; it also drops when the box reports an error
   #_w1 := #OUT.BQ10_CMD AND NOT #ONS.Pulse11;   // rising edge
   #ONS.Pulse11 := #OUT.BQ10_CMD;
   IF #_w1 THEN #FP_PARM.BQ10_CNT := #FP_PARM.BQ10_CNT + 1; END_IF;
   IF #FP_PARM.BQ10_CNT_RST THEN #FP_PARM.BQ10_CNT := 0; END_IF;
   #DummyBool := #_w1 AND #FP_PARM.BQ10_CNT_RST;
END_REGION

REGION Network 90: Blast Counter 11
   // ENO of a box is taken as its EN; it also drops when the box reports an error
   #_w1 := #OUT.BQ11_CMD AND NOT #ONS.Pulse12;   // rising edge
   #ONS.Pulse12 := #OUT.BQ11_CMD;
   IF #_w1 THEN #FP_PARM.BQ11_CNT := #FP_PARM.BQ11_CNT + 1; END_IF;
   IF #FP_PARM.BQ11_CNT_RST THEN #FP_PARM.BQ11_CNT := 0; END_IF;
   #DummyBool := #_w1 AND #FP_PARM.BQ11_CNT_RST;
END_REGION

REGION Network 91: Blast Counter 12
   // ENO of a box is taken as its EN; it also drops when the box reports an error
   #_w1 := #OUT.BQ12_CMD AND NOT #ONS.Pulse13;   // rising edge
   #ONS.Pulse13 := #OUT.BQ12_CMD;
   IF #_w1 THEN #FP_PARM.BQ12_CNT := #FP_PARM.BQ12_CNT + 1; END_IF;
   IF #FP_PARM.BQ12_CNT_RST THEN #FP_PARM.BQ12_CNT := 0; END_IF;
   #DummyBool := #_w1 AND #FP_PARM.BQ12_CNT_RST;
END_REGION

REGION Network 92: Blast Counter 13
   // ENO of a box is taken as its EN; it also drops when the box reports an error
   #_w1 := #OUT.BQ13_CMD AND NOT #ONS.Pulse14;   // rising edge
   #ONS.Pulse14 := #OUT.BQ13_CMD;
   IF #_w1 THEN #FP_PARM.BQ13_CNT := #FP_PARM.BQ13_CNT + 1; END_IF;
   IF #FP_PARM.BQ13_CNT_RST THEN #FP_PARM.BQ13_CNT := 0; END_IF;
   #DummyBool := #_w1 AND #FP_PARM.BQ13_CNT_RST;
END_REGION

REGION Network 93: Blast Counter 14
   // ENO of a box is taken as its EN; it also drops when the box reports an error
   #_w1 := #OUT.BQ14_CMD AND NOT #ONS.Pulse15;   // rising edge
   #ONS.Pulse15 := #OUT.BQ14_CMD;
   IF #_w1 THEN #FP_PARM.BQ14_CNT := #FP_PARM.BQ14_CNT + 1; END_IF;
   IF #FP_PARM.BQ14_CNT_RST THEN #FP_PARM.BQ14_CNT := 0; END_IF;
   #DummyBool := #_w1 AND #FP_PARM.BQ14_CNT_RST;
END_REGION

REGION Network 94: Blast Counter 15
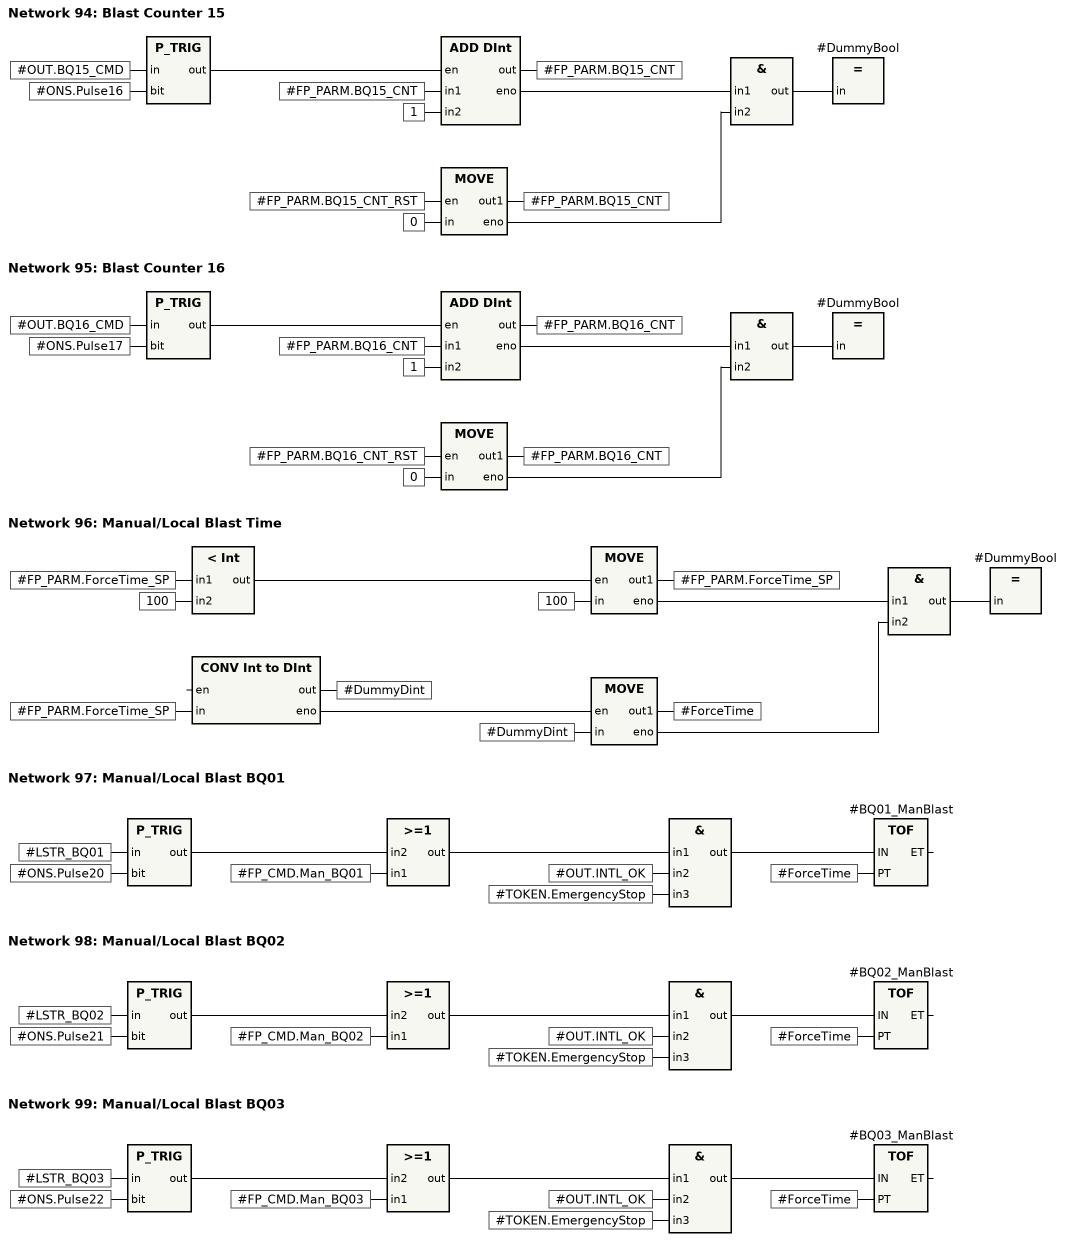
   // ENO of a box is taken as its EN; it also drops when the box reports an error
   #_w1 := #OUT.BQ15_CMD AND NOT #ONS.Pulse16;   // rising edge
   #ONS.Pulse16 := #OUT.BQ15_CMD;
   IF #_w1 THEN #FP_PARM.BQ15_CNT := #FP_PARM.BQ15_CNT + 1; END_IF;
   IF #FP_PARM.BQ15_CNT_RST THEN #FP_PARM.BQ15_CNT := 0; END_IF;
   #DummyBool := #_w1 AND #FP_PARM.BQ15_CNT_RST;
END_REGION

REGION Network 95: Blast Counter 16
   // ENO of a box is taken as its EN; it also drops when the box reports an error
   #_w1 := #OUT.BQ16_CMD AND NOT #ONS.Pulse17;   // rising edge
   #ONS.Pulse17 := #OUT.BQ16_CMD;
   IF #_w1 THEN #FP_PARM.BQ16_CNT := #FP_PARM.BQ16_CNT + 1; END_IF;
   IF #FP_PARM.BQ16_CNT_RST THEN #FP_PARM.BQ16_CNT := 0; END_IF;
   #DummyBool := #_w1 AND #FP_PARM.BQ16_CNT_RST;
END_REGION

REGION Network 96: Manual/Local Blast Time
   // Keep into range and typ cast
   // ENO of a box is taken as its EN; it also drops when the box reports an error
   #_w1 := #FP_PARM.ForceTime_SP < 100;
   IF #_w1 THEN #FP_PARM.ForceTime_SP := 100; END_IF;
   #DummyDint := INT_TO_DINT(#FP_PARM.ForceTime_SP);
   #ForceTime := #DummyDint;
   #DummyBool := #_w1;
END_REGION

REGION Network 97: Manual/Local Blast BQ01
   #_w1 := #LSTR_BQ01 AND NOT #ONS.Pulse20;   // rising edge
   #ONS.Pulse20 := #LSTR_BQ01;
   #BQ01_ManBlast(IN := (#_w1 OR #FP_CMD.Man_BQ01) AND #OUT.INTL_OK AND #TOKEN.EmergencyStop, PT := #ForceTime);   // TOF
END_REGION

REGION Network 98: Manual/Local Blast BQ02
   #_w1 := #LSTR_BQ02 AND NOT #ONS.Pulse21;   // rising edge
   #ONS.Pulse21 := #LSTR_BQ02;
   #BQ02_ManBlast(IN := (#_w1 OR #FP_CMD.Man_BQ02) AND #OUT.INTL_OK AND #TOKEN.EmergencyStop, PT := #ForceTime);   // TOF
END_REGION

REGION Network 99: Manual/Local Blast BQ03
   #_w1 := #LSTR_BQ03 AND NOT #ONS.Pulse22;   // rising edge
   #ONS.Pulse22 := #LSTR_BQ03;
   #BQ03_ManBlast(IN := (#_w1 OR #FP_CMD.Man_BQ03) AND #OUT.INTL_OK AND #TOKEN.EmergencyStop, PT := #ForceTime);   // TOF
END_REGION

REGION Network 100: Manual/Local Blast BQ04
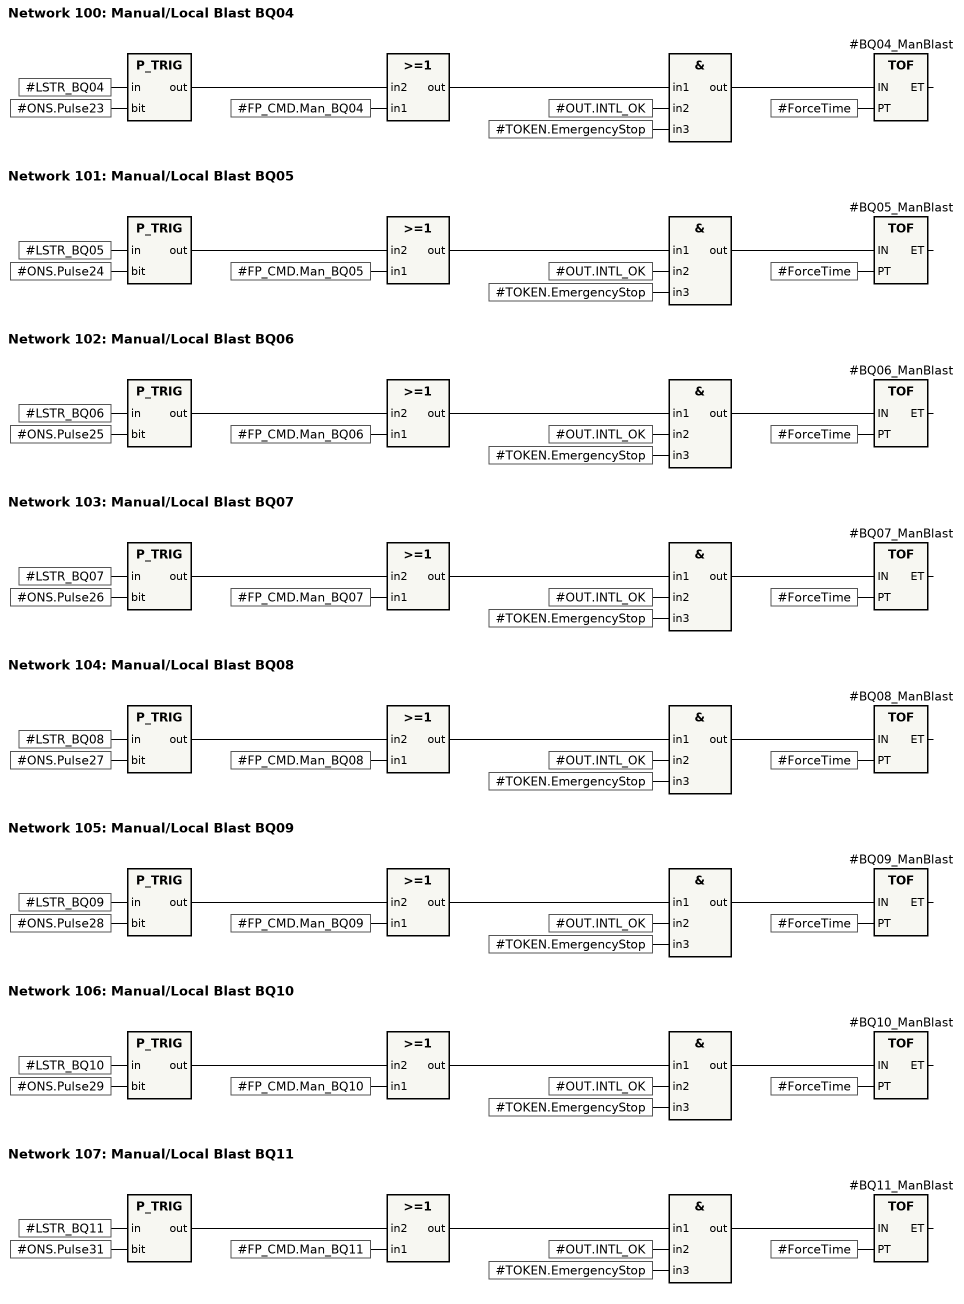
   #_w1 := #LSTR_BQ04 AND NOT #ONS.Pulse23;   // rising edge
   #ONS.Pulse23 := #LSTR_BQ04;
   #BQ04_ManBlast(IN := (#_w1 OR #FP_CMD.Man_BQ04) AND #OUT.INTL_OK AND #TOKEN.EmergencyStop, PT := #ForceTime);   // TOF
END_REGION

REGION Network 101: Manual/Local Blast BQ05
   #_w1 := #LSTR_BQ05 AND NOT #ONS.Pulse24;   // rising edge
   #ONS.Pulse24 := #LSTR_BQ05;
   #BQ05_ManBlast(IN := (#_w1 OR #FP_CMD.Man_BQ05) AND #OUT.INTL_OK AND #TOKEN.EmergencyStop, PT := #ForceTime);   // TOF
END_REGION

REGION Network 102: Manual/Local Blast BQ06
   #_w1 := #LSTR_BQ06 AND NOT #ONS.Pulse25;   // rising edge
   #ONS.Pulse25 := #LSTR_BQ06;
   #BQ06_ManBlast(IN := (#_w1 OR #FP_CMD.Man_BQ06) AND #OUT.INTL_OK AND #TOKEN.EmergencyStop, PT := #ForceTime);   // TOF
END_REGION

REGION Network 103: Manual/Local Blast BQ07
   #_w1 := #LSTR_BQ07 AND NOT #ONS.Pulse26;   // rising edge
   #ONS.Pulse26 := #LSTR_BQ07;
   #BQ07_ManBlast(IN := (#_w1 OR #FP_CMD.Man_BQ07) AND #OUT.INTL_OK AND #TOKEN.EmergencyStop, PT := #ForceTime);   // TOF
END_REGION

REGION Network 104: Manual/Local Blast BQ08
   #_w1 := #LSTR_BQ08 AND NOT #ONS.Pulse27;   // rising edge
   #ONS.Pulse27 := #LSTR_BQ08;
   #BQ08_ManBlast(IN := (#_w1 OR #FP_CMD.Man_BQ08) AND #OUT.INTL_OK AND #TOKEN.EmergencyStop, PT := #ForceTime);   // TOF
END_REGION

REGION Network 105: Manual/Local Blast BQ09
   #_w1 := #LSTR_BQ09 AND NOT #ONS.Pulse28;   // rising edge
   #ONS.Pulse28 := #LSTR_BQ09;
   #BQ09_ManBlast(IN := (#_w1 OR #FP_CMD.Man_BQ09) AND #OUT.INTL_OK AND #TOKEN.EmergencyStop, PT := #ForceTime);   // TOF
END_REGION

REGION Network 106: Manual/Local Blast BQ10
   #_w1 := #LSTR_BQ10 AND NOT #ONS.Pulse29;   // rising edge
   #ONS.Pulse29 := #LSTR_BQ10;
   #BQ10_ManBlast(IN := (#_w1 OR #FP_CMD.Man_BQ10) AND #OUT.INTL_OK AND #TOKEN.EmergencyStop, PT := #ForceTime);   // TOF
END_REGION

REGION Network 107: Manual/Local Blast BQ11
   #_w1 := #LSTR_BQ11 AND NOT #ONS.Pulse31;   // rising edge
   #ONS.Pulse31 := #LSTR_BQ11;
   #BQ11_ManBlast(IN := (#_w1 OR #FP_CMD.Man_BQ11) AND #OUT.INTL_OK AND #TOKEN.EmergencyStop, PT := #ForceTime);   // TOF
END_REGION

REGION Network 108: Manual/Local Blast BQ12
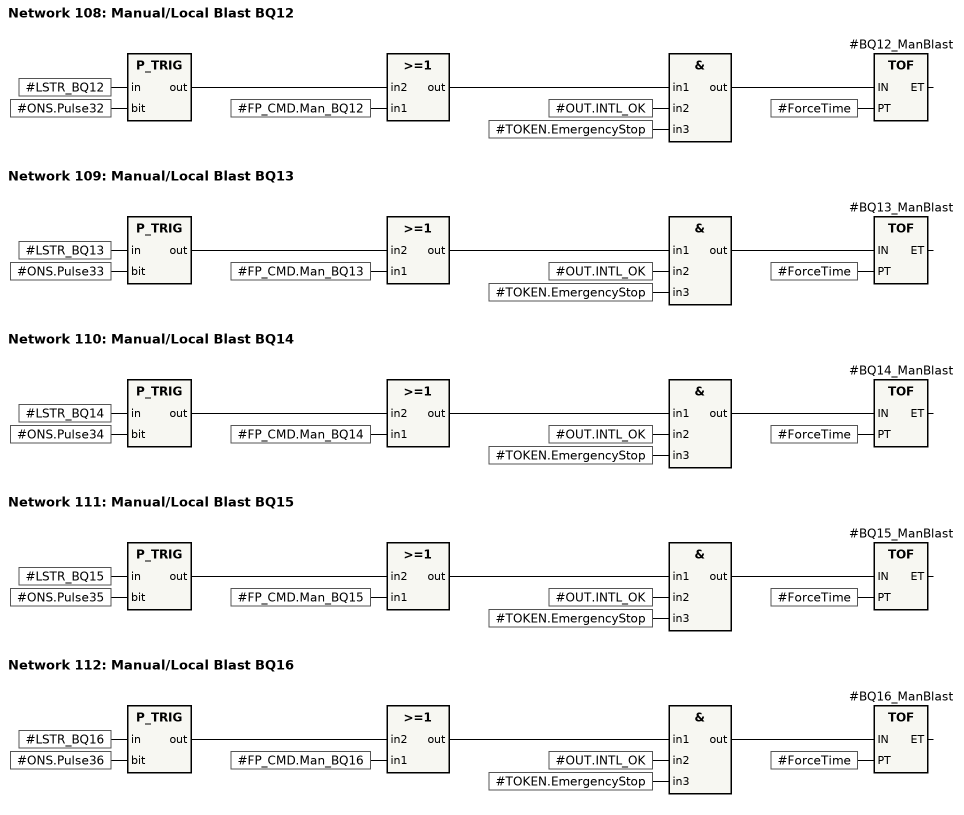
   #_w1 := #LSTR_BQ12 AND NOT #ONS.Pulse32;   // rising edge
   #ONS.Pulse32 := #LSTR_BQ12;
   #BQ12_ManBlast(IN := (#_w1 OR #FP_CMD.Man_BQ12) AND #OUT.INTL_OK AND #TOKEN.EmergencyStop, PT := #ForceTime);   // TOF
END_REGION

REGION Network 109: Manual/Local Blast BQ13
   #_w1 := #LSTR_BQ13 AND NOT #ONS.Pulse33;   // rising edge
   #ONS.Pulse33 := #LSTR_BQ13;
   #BQ13_ManBlast(IN := (#_w1 OR #FP_CMD.Man_BQ13) AND #OUT.INTL_OK AND #TOKEN.EmergencyStop, PT := #ForceTime);   // TOF
END_REGION

REGION Network 110: Manual/Local Blast BQ14
   #_w1 := #LSTR_BQ14 AND NOT #ONS.Pulse34;   // rising edge
   #ONS.Pulse34 := #LSTR_BQ14;
   #BQ14_ManBlast(IN := (#_w1 OR #FP_CMD.Man_BQ14) AND #OUT.INTL_OK AND #TOKEN.EmergencyStop, PT := #ForceTime);   // TOF
END_REGION

REGION Network 111: Manual/Local Blast BQ15
   #_w1 := #LSTR_BQ15 AND NOT #ONS.Pulse35;   // rising edge
   #ONS.Pulse35 := #LSTR_BQ15;
   #BQ15_ManBlast(IN := (#_w1 OR #FP_CMD.Man_BQ15) AND #OUT.INTL_OK AND #TOKEN.EmergencyStop, PT := #ForceTime);   // TOF
END_REGION

REGION Network 112: Manual/Local Blast BQ16
   #_w1 := #LSTR_BQ16 AND NOT #ONS.Pulse36;   // rising edge
   #ONS.Pulse36 := #LSTR_BQ16;
   #BQ16_ManBlast(IN := (#_w1 OR #FP_CMD.Man_BQ16) AND #OUT.INTL_OK AND #TOKEN.EmergencyStop, PT := #ForceTime);   // TOF
END_REGION

REGION Network 113: Reset Faceplate Commands
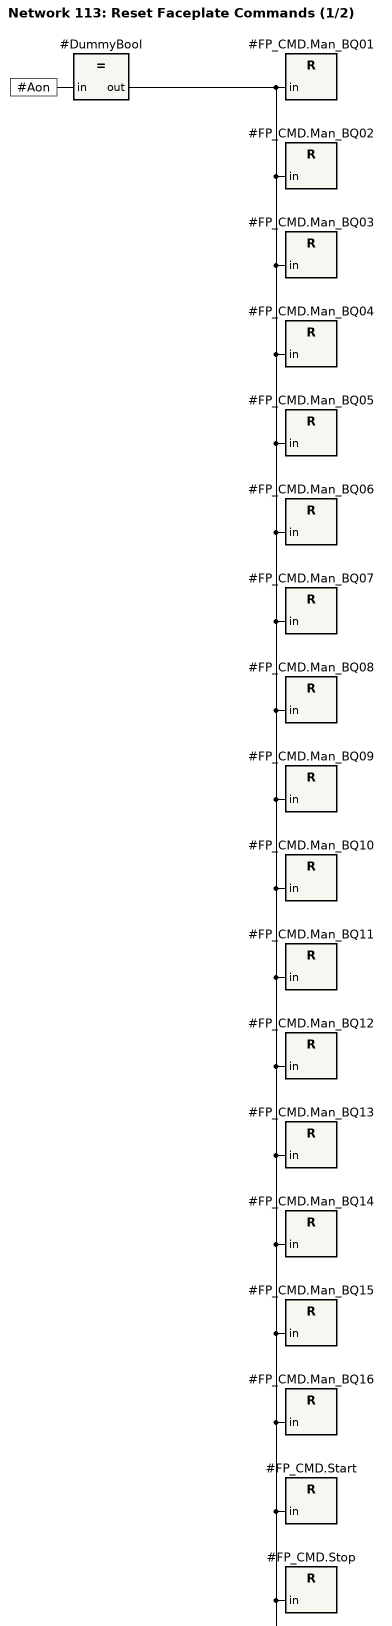
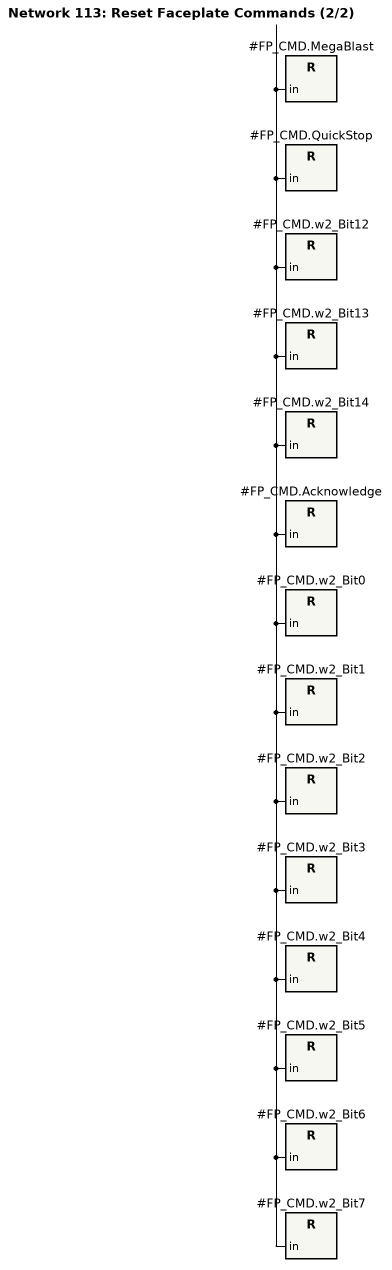
   #DummyBool := #Aon;
   IF #Aon THEN
       #FP_CMD.Man_BQ01 := FALSE;
       #FP_CMD.Man_BQ02 := FALSE;
       #FP_CMD.Man_BQ03 := FALSE;
       #FP_CMD.Man_BQ04 := FALSE;
       #FP_CMD.Man_BQ05 := FALSE;
       #FP_CMD.Man_BQ06 := FALSE;
       #FP_CMD.Man_BQ07 := FALSE;
       #FP_CMD.Man_BQ08 := FALSE;
       #FP_CMD.Man_BQ09 := FALSE;
       #FP_CMD.Man_BQ10 := FALSE;
       #FP_CMD.Man_BQ11 := FALSE;
       #FP_CMD.Man_BQ12 := FALSE;
       #FP_CMD.Man_BQ13 := FALSE;
       #FP_CMD.Man_BQ14 := FALSE;
       #FP_CMD.Man_BQ15 := FALSE;
       #FP_CMD.Man_BQ16 := FALSE;
       #FP_CMD.Start := FALSE;
       #FP_CMD.Stop := FALSE;
       #FP_CMD.MegaBlast := FALSE;
       #FP_CMD.QuickStop := FALSE;
       #FP_CMD.w2_Bit12 := FALSE;
       #FP_CMD.w2_Bit13 := FALSE;
       #FP_CMD.w2_Bit14 := FALSE;
       #FP_CMD.Acknowledge := FALSE;
       #FP_CMD.w2_Bit0 := FALSE;
       #FP_CMD.w2_Bit1 := FALSE;
       #FP_CMD.w2_Bit2 := FALSE;
       #FP_CMD.w2_Bit3 := FALSE;
       #FP_CMD.w2_Bit4 := FALSE;
       #FP_CMD.w2_Bit5 := FALSE;
       #FP_CMD.w2_Bit6 := FALSE;
       #FP_CMD.w2_Bit7 := FALSE;
   END_IF;
END_REGION

REGION Network 114: Reset Faceplate Commands
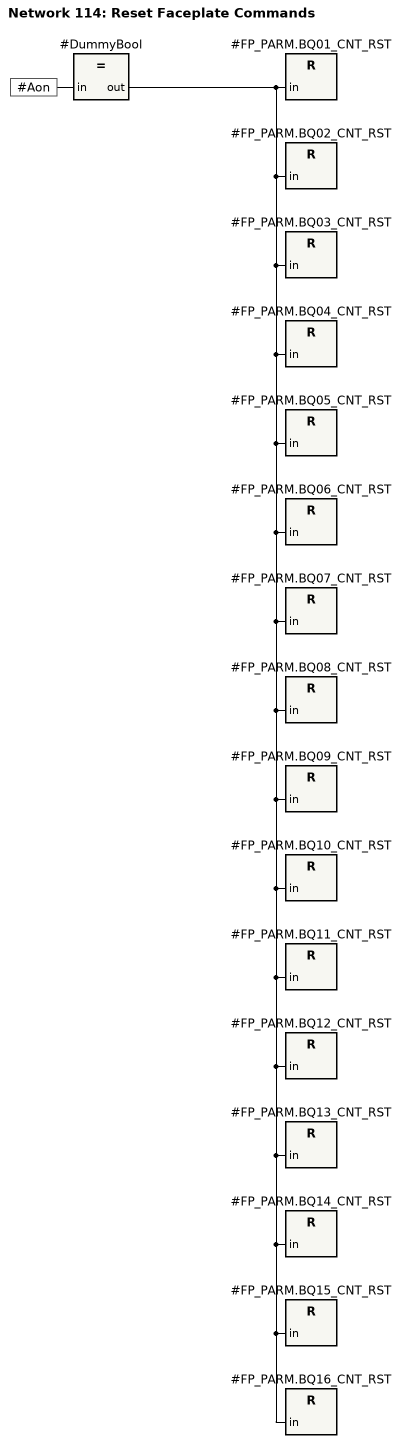
   #DummyBool := #Aon;
   IF #Aon THEN
       #FP_PARM.BQ01_CNT_RST := FALSE;
       #FP_PARM.BQ02_CNT_RST := FALSE;
       #FP_PARM.BQ03_CNT_RST := FALSE;
       #FP_PARM.BQ04_CNT_RST := FALSE;
       #FP_PARM.BQ05_CNT_RST := FALSE;
       #FP_PARM.BQ06_CNT_RST := FALSE;
       #FP_PARM.BQ07_CNT_RST := FALSE;
       #FP_PARM.BQ08_CNT_RST := FALSE;
       #FP_PARM.BQ09_CNT_RST := FALSE;
       #FP_PARM.BQ10_CNT_RST := FALSE;
       #FP_PARM.BQ11_CNT_RST := FALSE;
       #FP_PARM.BQ12_CNT_RST := FALSE;
       #FP_PARM.BQ13_CNT_RST := FALSE;
       #FP_PARM.BQ14_CNT_RST := FALSE;
       #FP_PARM.BQ15_CNT_RST := FALSE;
       #FP_PARM.BQ16_CNT_RST := FALSE;
   END_IF;
END_REGION

REGION Network 115: Old Program SP
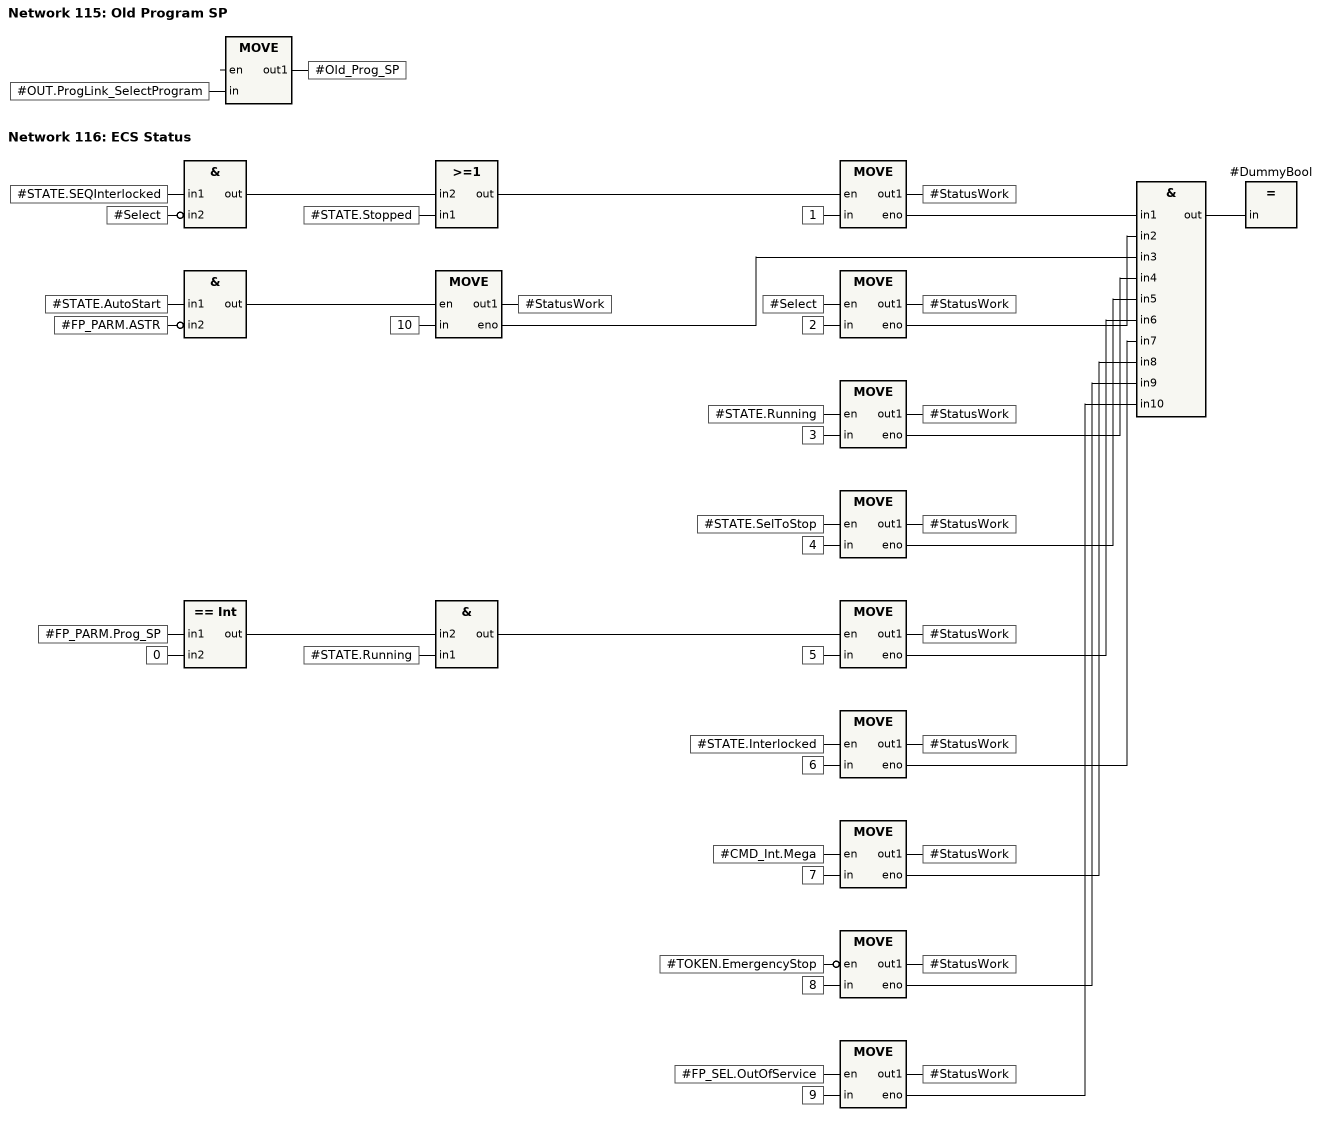
   #Old_Prog_SP := #OUT.ProgLink_SelectProgram;
END_REGION

REGION Network 116: ECS Status
   // 1)  Stopped
   // 2)  Start Selected
   // 3)  Running
   // 4)  Stop Selected                                                        
   // 5)  Running No Program Selected
   // 6)  Interlocked
   // 7)  Mega Blast
   // 8)  Emergency Stop
   // 9)  Out of Service
   // 10) Interval Start
   // 
   // 
   // Build 003-11 Aug 2021- SURAM-IN- Interval Start Status Work Derived
   // ENO of a box is taken as its EN; it also drops when the box reports an error
   #_w1 := (#STATE.SEQInterlocked AND NOT #Select) OR #STATE.Stopped;
   IF #_w1 THEN #StatusWork := 1; END_IF;
   IF #Select THEN #StatusWork := 2; END_IF;
   #_w2 := #STATE.AutoStart AND NOT #FP_PARM.ASTR;
   IF #_w2 THEN #StatusWork := 10; END_IF;
   IF #STATE.Running THEN #StatusWork := 3; END_IF;
   IF #STATE.SelToStop THEN #StatusWork := 4; END_IF;
   #_w3 := (#FP_PARM.Prog_SP = 0) AND #STATE.Running;
   IF #_w3 THEN #StatusWork := 5; END_IF;
   IF #STATE.Interlocked THEN #StatusWork := 6; END_IF;
   IF #CMD_Int.Mega THEN #StatusWork := 7; END_IF;
   IF NOT #TOKEN.EmergencyStop THEN #StatusWork := 8; END_IF;
   IF #FP_SEL.OutOfService THEN #StatusWork := 9; END_IF;
   #DummyBool := #_w1 AND #Select AND #_w2 AND #STATE.Running AND #STATE.SelToStop AND #_w3 AND #STATE.Interlocked AND #CMD_Int.Mega AND NOT #TOKEN.EmergencyStop AND #FP_SEL.OutOfService;
END_REGION

REGION Network 117: Extended Status
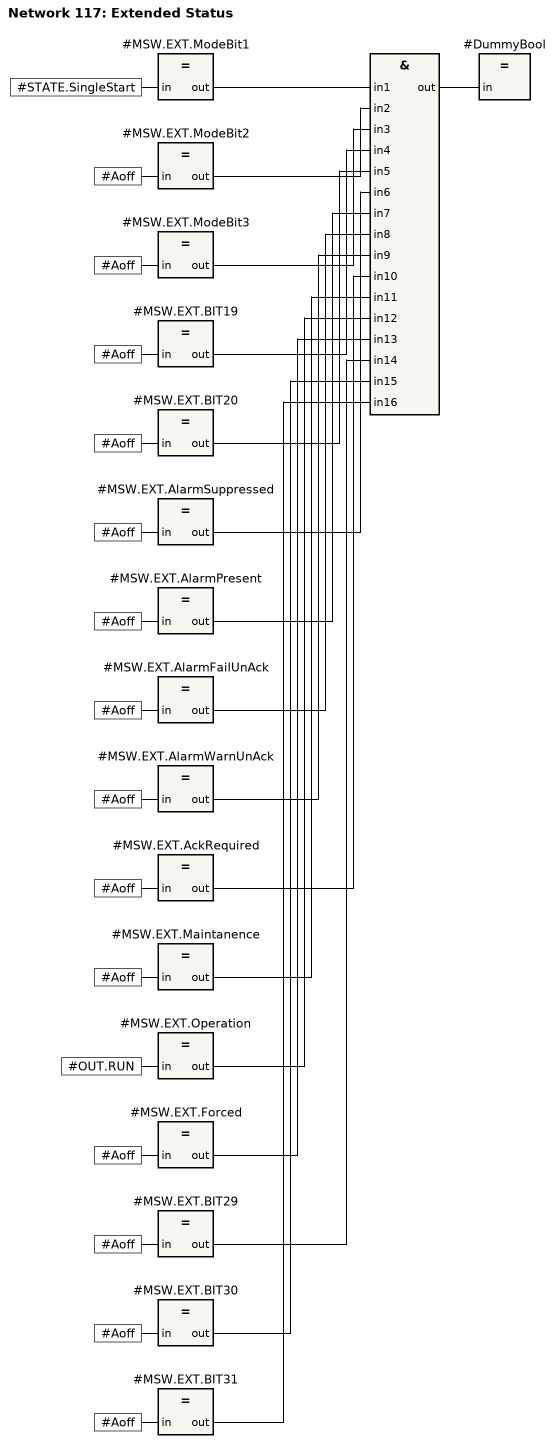
   #MSW.EXT.ModeBit1 := #STATE.SingleStart;
   #MSW.EXT.ModeBit2 := #Aoff;
   #MSW.EXT.ModeBit3 := #Aoff;
   #MSW.EXT.BIT19 := #Aoff;
   #MSW.EXT.BIT20 := #Aoff;
   #MSW.EXT.AlarmSuppressed := #Aoff;
   #MSW.EXT.AlarmPresent := #Aoff;
   #MSW.EXT.AlarmFailUnAck := #Aoff;
   #MSW.EXT.AlarmWarnUnAck := #Aoff;
   #MSW.EXT.AckRequired := #Aoff;
   #MSW.EXT.Maintanence := #Aoff;
   #MSW.EXT.Operation := #OUT.RUN;
   #MSW.EXT.Forced := #Aoff;
   #MSW.EXT.BIT29 := #Aoff;
   #MSW.EXT.BIT30 := #Aoff;
   #MSW.EXT.BIT31 := #Aoff;
   #DummyBool := #STATE.SingleStart AND #Aoff AND #Aoff AND #Aoff AND #Aoff AND #Aoff AND #Aoff AND #Aoff AND #Aoff AND #Aoff AND #Aoff AND #OUT.RUN AND #Aoff AND #Aoff AND #Aoff AND #Aoff;
END_REGION

REGION Network 118: Update Internal MSW and Timestamp
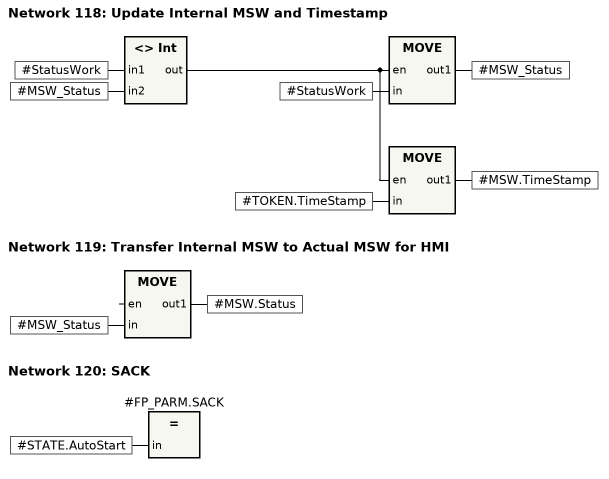
   #_w1 := #StatusWork <> #MSW_Status;
   IF #_w1 THEN
       #MSW_Status := #StatusWork;
       #MSW.TimeStamp := #TOKEN.TimeStamp;
   END_IF;
END_REGION

REGION Network 119: Transfer Internal MSW to Actual MSW for HMI
   #MSW.Status := #MSW_Status;
END_REGION

REGION Network 120: SACK
   // Build 003-11 Aug 2021- SURAM-IN- State Autostart moved to SACK logic derived
   #FP_PARM.SACK := #STATE.AutoStart;
END_REGION

REGION Network 121: Update Token Data
   // Build 002 - 24.Jun.2020 (MIA-US): Replace "Select" with "SEL" in the TOKEN.SACK_On logic
   // Build 003-11 Aug 2021- SURAM-IN- State Running replaced with State Autostart
